LIN {X 0,Y 335.308,Z 623.747,A -85,B 0,C 180,E1 -19732.854,E2 -19732.854} C_VEL
LIN {X 0,Y 329.002,Z 618.791,A -85,B 0,C 180,E1 -19734.521,E2 -19734.521} C_VEL
LIN {X 0,Y 320.046,Z 611.53,A -85,B 0,C 180,E1 -19736.705,E2 -19736.705} C_VEL
LIN {X 0,Y 311.713,Z 604.517,A -85,B 0,C 180,E1 -19738.536,E2 -19738.536} C_VEL
LIN {X 0,Y 303.671,Z 597.573,A -85,B 0,C 180,E1 -19740.106,E2 -19740.106} C_VEL
LIN {X 0,Y 294.083,Z 589.042,A -85,B 0,C 180,E1 -19741.756,E2 -19741.756} C_VEL
LIN {X 0,Y 277.911,Z 573.415,A -85,B 0,C 180,E1 -19744.368,E2 -19744.368} C_VEL
LIN {X 0,Y 267.025,Z 560.92,A -85,B 0,C 180,E1 -19746.403,E2 -19746.403} C_VEL
LIN {X 0,Y 258.838,Z 549.026,A -85,B 0,C 180,E1 -19748.172,E2 -19748.172} C_VEL
LIN {X 0,Y 247.972,Z 530.618,A -85,B 0,C 180,E1 -19750.877,E2 -19750.877} C_VEL
LIN {X 0,Y 240.07,Z 518.715,A -85,B 0,C 180,E1 -19753.019,E2 -19753.019} C_VEL
LIN {X 0,Y 237.499,Z 514.891,A -85,B 0,C 180,E1 -19753.761,E2 -19753.761} C_VEL
LIN {X 0,Y 235.646,Z 512.583,A -85,B 0,C 180,E1 -19754.294,E2 -19754.294} C_VEL
LIN {X 0,Y 235.056,Z 510.889,A -85,B 0,C 180,E1 -19754.626,E2 -19754.626} C_VEL
LIN {X 0,Y 234.948,Z 510.343,A -85,B 0,C 180,E1 -19755.075,E2 -19755.075} C_VEL
LIN {X 0,Y 234.945,Z 510.328,A -85,B 0,C 180,E1 -19758.847,E2 -19758.847} C_VEL
LIN {X 0,Y 234.94,Z 510.326,A -85,B 0,C 180,E1 -19763.254,E2 -19763.254} C_VEL
LIN {X 0,Y 234.955,Z 510.335,A -85,B 0,C 180,E1 -19767.425,E2 -19767.425} C_VEL
LIN {X 0,Y 234.947,Z 510.334,A -85,B 0,C 180,E1 -19771.406,E2 -19771.406} C_VEL
LIN {X 0,Y 234.981,Z 510.31,A -85,B 0,C 180,E1 -19775.247,E2 -19775.247} C_VEL
LIN {X 0,Y 235.006,Z 510.337,A -85,B 0,C 180,E1 -19778.97,E2 -19778.97} C_VEL
LIN {X 0,Y 235.09,Z 510.293,A -85,B 0,C 180,E1 -19783.061,E2 -19783.061} C_VEL
LIN {X 0,Y 235.108,Z 510.307,A -85,B 0,C 180,E1 -19787.923,E2 -19787.923} C_VEL
LIN {X 0,Y 235.326,Z 510.265,A -85,B 0,C 180,E1 -19791.413,E2 -19791.413} C_VEL
LIN {X 0,Y 235.369,Z 510.285,A -85,B 0,C 180,E1 -19793.141,E2 -19793.141} C_VEL
LIN {X 0,Y 235.59,Z 510.222,A -85,B 0,C 180,E1 -19798.291,E2 -19798.291} C_VEL
LIN {X 0,Y 235.591,Z 510.26,A -85,B 0,C 180,E1 -19801.71,E2 -19801.71} C_VEL
LIN {X 0,Y 235.398,Z 510.252,A -85,B 0,C 180,E1 -19806.86,E2 -19806.86} C_VEL
LIN {X 0,Y 235.234,Z 510.306,A -85,B 0,C 180,E1 -19810.327,E2 -19810.327} C_VEL
LIN {X 0,Y 235.108,Z 510.306,A -85,B 0,C 180,E1 -19815.608,E2 -19815.608} C_VEL
LIN {X 0,Y 235.003,Z 510.313,A -85,B 0,C 180,E1 -19819.207,E2 -19819.207} C_VEL
LIN {X 0,Y 234.949,Z 510.333,A -85,B 0,C 180,E1 -19822.885,E2 -19822.885} C_VEL
LIN {X 0,Y 234.964,Z 510.315,A -85,B 0,C 180,E1 -19826.659,E2 -19826.659} C_VEL
LIN {X 0,Y 234.92,Z 510.347,A -85,B 0,C 180,E1 -19830.57,E2 -19830.57} C_VEL
LIN {X 0,Y 234.959,Z 510.33,A -85,B 0,C 180,E1 -19834.634,E2 -19834.634} C_VEL
LIN {X 0,Y 234.966,Z 510.331,A -85,B 0,C 180,E1 -19838.953,E2 -19838.953} C_VEL
LIN {X 0,Y 234.951,Z 510.537,A -85,B 0,C 180,E1 -19842.193,E2 -19842.193} C_VEL
LIN {X 0,Y 236.478,Z 516.25,A -85,B 0,C 180,E1 -19845.577,E2 -19845.577} C_VEL
LIN {X 0,Y 238.772,Z 520.508,A -85,B 0,C 180,E1 -19846.368,E2 -19846.368} C_VEL
LIN {X 0,Y 243.465,Z 528.613,A -85,B 0,C 180,E1 -19847.722,E2 -19847.722} C_VEL
LIN {X 0,Y 249.61,Z 540.017,A -85,B 0,C 180,E1 -19849.406,E2 -19849.406} C_VEL
LIN {X 0,Y 256.246,Z 553.836,A -85,B 0,C 180,E1 -19851.145,E2 -19851.145} C_VEL
LIN {X 0,Y 261.647,Z 566.971,A -85,B 0,C 180,E1 -19852.53,E2 -19852.53} C_VEL
LIN {X 0,Y 262.847,Z 573.625,A -85,B 0,C 180,E1 -19852.952,E2 -19852.952} C_VEL
LIN {X 0,Y 262.9,Z 576.826,A -85,B 0,C 180,E1 -19853.067,E2 -19853.067} C_VEL
LIN {X 0,Y 261.778,Z 581.327,A -85,B 0,C 180,E1 -19853.035,E2 -19853.035} C_VEL
LIN {X 0,Y 258.338,Z 590.232,A -85,B 0,C 180,E1 -19852.767,E2 -19852.767} C_VEL
LIN {X 0,Y 257.612,Z 594.257,A -85,B 0,C 180,E1 -19852.783,E2 -19852.783} C_VEL
LIN {X 0,Y 254.782,Z 653.012,A -85,B 0,C 180,E1 -19854.378,E2 -19854.378} C_VEL
LIN {X 0,Y 253.718,Z 664.354,A -85,B 0,C 180,E1 -19854.856,E2 -19854.856} C_VEL
LIN {X 0,Y 252.166,Z 675.789,A -85,B 0,C 180,E1 -19855.521,E2 -19855.521} C_VEL
LIN {X 0,Y 250.179,Z 687.439,A -85,B 0,C 180,E1 -19856.424,E2 -19856.424} C_VEL
LIN {X 0,Y 247.382,Z 701.15,A -85,B 0,C 180,E1 -19857.814,E2 -19857.814} C_VEL
LIN {X 0,Y 244.332,Z 713.482,A -85,B 0,C 180,E1 -19859.472,E2 -19859.472} C_VEL
LIN {X 0,Y 241.782,Z 723.247,A -85,B 0,C 180,E1 -19861.103,E2 -19861.103} C_VEL
LIN {X 0,Y 239.044,Z 732.264,A -85,B 0,C 180,E1 -19862.89,E2 -19862.89} C_VEL
LIN {X 0,Y 236.794,Z 739.236,A -85,B 0,C 180,E1 -19864.51,E2 -19864.51} C_VEL
LIN {X 0,Y 234.414,Z 746.76,A -85,B 0,C 180,E1 -19866.594,E2 -19866.594} C_VEL
LIN {X 0,Y 232.273,Z 753.234,A -85,B 0,C 180,E1 -19868.71,E2 -19868.71} C_VEL
LIN {X 0,Y 230.021,Z 760.213,A -85,B 0,C 180,E1 -19871.499,E2 -19871.499} C_VEL
LIN {X 0,Y 228.524,Z 765.213,A -85,B 0,C 180,E1 -19873.932,E2 -19873.932} C_VEL
LIN {X 0,Y 227.23,Z 769.661,A -85,B 0,C 180,E1 -19876.587,E2 -19876.587} C_VEL
LIN {X 0,Y 226.362,Z 773.212,A -85,B 0,C 180,E1 -19879.264,E2 -19879.264} C_VEL
LIN {X 0,Y 225.99,Z 775.156,A -85,B 0,C 180,E1 -19881.055,E2 -19881.055} C_VEL
LIN {X 0,Y 225.644,Z 777.85,A -85,B 0,C 180,E1 -19884.639,E2 -19884.639} C_VEL
LIN {X 0,Y 225.64,Z 779.149,A -85,B 0,C 180,E1 -19888.215,E2 -19888.215} C_VEL
LIN {X 0,Y 225.716,Z 779.404,A -85,B 0,C 180,E1 -19890,E2 -19890} C_VEL
LIN {X 0,Y 225.584,Z 778.671,A -85,B 0,C 180,E1 -19893.572,E2 -19893.572} C_VEL
LIN {X 0,Y 225.644,Z 777.85,A -85,B 0,C 180,E1 -19895.361,E2 -19895.361} C_VEL
LIN {X 0,Y 225.99,Z 775.156,A -85,B 0,C 180,E1 -19898.945,E2 -19898.945} C_VEL
LIN {X 0,Y 226.591,Z 772.193,A -85,B 0,C 180,E1 -19901.631,E2 -19901.631} C_VEL
LIN {X 0,Y 227.632,Z 768.363,A -85,B 0,C 180,E1 -19904.299,E2 -19904.299} C_VEL
LIN {X 0,Y 229.041,Z 763.597,A -85,B 0,C 180,E1 -19906.948,E2 -19906.948} C_VEL
LIN {X 0,Y 231.158,Z 756.648,A -85,B 0,C 180,E1 -19910.001,E2 -19910.001} C_VEL
LIN {X 0,Y 233.077,Z 750.772,A -85,B 0,C 180,E1 -19912.142,E2 -19912.142} C_VEL
LIN {X 0,Y 235.796,Z 742.36,A -85,B 0,C 180,E1 -19914.662,E2 -19914.662} C_VEL
LIN {X 0,Y 237.911,Z 735.901,A -85,B 0,C 180,E1 -19916.302,E2 -19916.302} C_VEL
LIN {X 0,Y 240.892,Z 726.426,A -85,B 0,C 180,E1 -19918.3,E2 -19918.3} C_VEL
LIN {X 0,Y 243.327,Z 717.587,A -85,B 0,C 180,E1 -19919.875,E2 -19919.875} C_VEL
LIN {X 0,Y 245.614,Z 708.498,A -85,B 0,C 180,E1 -19921.239,E2 -19921.239} C_VEL
LIN {X 0,Y 248.097,Z 697.694,A -85,B 0,C 180,E1 -19922.562,E2 -19922.562} C_VEL
LIN {X 0,Y 250.187,Z 687.44,A -85,B 0,C 180,E1 -19923.575,E2 -19923.575} C_VEL
LIN {X 0,Y 251.97,Z 677.149,A -85,B 0,C 180,E1 -19924.389,E2 -19924.389} C_VEL
LIN {X 0,Y 253.609,Z 665.266,A -85,B 0,C 180,E1 -19925.1,E2 -19925.1} C_VEL
LIN {X 0,Y 254.706,Z 653.918,A -85,B 0,C 180,E1 -19925.59,E2 -19925.59} C_VEL
LIN {X 0,Y 256.027,Z 629.639,A -85,B 0,C 180,E1 -19926.273,E2 -19926.273} C_VEL
LIN {X 0,Y 258.131,Z 580.661,A -85,B 0,C 180,E1 -19927.595,E2 -19927.595} C_VEL
LIN {X 0,Y 256.026,Z 569.105,A -85,B 0,C 180,E1 -19928.359,E2 -19928.359} C_VEL
LIN {X 0,Y 249.816,Z 554.326,A -85,B 0,C 180,E1 -19930.027,E2 -19930.027} C_VEL
LIN {X 0,Y 243.956,Z 542.258,A -85,B 0,C 180,E1 -19931.647,E2 -19931.647} C_VEL
LIN {X 0,Y 237.336,Z 529.983,A -85,B 0,C 180,E1 -19933.573,E2 -19933.573} C_VEL
LIN {X 0,Y 231.653,Z 520.434,A -85,B 0,C 180,E1 -19935.326,E2 -19935.326} C_VEL
LIN {X 0,Y 229.167,Z 516.078,A -85,B 0,C 180,E1 -19936.215,E2 -19936.215} C_VEL
LIN {X 0,Y 228.519,Z 513.68,A -85,B 0,C 180,E1 -19937.569,E2 -19937.569} C_VEL
LIN {X 0,Y 227.869,Z 511.239,A -85,B 0,C 180,E1 -19939.359,E2 -19939.359} C_VEL
LIN {X 0,Y 227.9,Z 511.223,A -85,B 0,C 180,E1 -19944.131,E2 -19944.131} C_VEL
LIN {X 0,Y 227.867,Z 511.211,A -85,B 0,C 180,E1 -19948.376,E2 -19948.376} C_VEL
LIN {X 0,Y 227.875,Z 511.196,A -85,B 0,C 180,E1 -19952.443,E2 -19952.443} C_VEL
LIN {X 0,Y 227.903,Z 511.221,A -85,B 0,C 180,E1 -19956.365,E2 -19956.365} C_VEL
LIN {X 0,Y 227.933,Z 511.187,A -85,B 0,C 180,E1 -19960.173,E2 -19960.173} C_VEL
LIN {X 0,Y 228.053,Z 511.194,A -85,B 0,C 180,E1 -19963.897,E2 -19963.897} C_VEL
LIN {X 0,Y 228.069,Z 511.167,A -85,B 0,C 180,E1 -19967.542,E2 -19967.542} C_VEL
LIN {X 0,Y 228.301,Z 511.167,A -85,B 0,C 180,E1 -19971.145,E2 -19971.145} C_VEL
LIN {X 0,Y 228.349,Z 511.132,A -85,B 0,C 180,E1 -19972.928,E2 -19972.928} C_VEL
LIN {X 0,Y 228.549,Z 511.138,A -85,B 0,C 180,E1 -19978.237,E2 -19978.237} C_VEL
LIN {X 0,Y 228.549,Z 511.098,A -85,B 0,C 180,E1 -19981.761,E2 -19981.761} C_VEL
LIN {X 0,Y 228.318,Z 511.16,A -85,B 0,C 180,E1 -19987.072,E2 -19987.072} C_VEL
LIN {X 0,Y 228.14,Z 511.155,A -85,B 0,C 180,E1 -19990.651,E2 -19990.651} C_VEL
LIN {X 0,Y 228.054,Z 511.201,A -85,B 0,C 180,E1 -19994.272,E2 -19994.272} C_VEL
LIN {X 0,Y 227.997,Z 511.176,A -85,B 0,C 180,E1 -19997.953,E2 -19997.953} C_VEL
LIN {X 0,Y 227.924,Z 511.204,A -85,B 0,C 180,E1 -20002.328,E2 -20002.328} C_VEL
LIN {X 0,Y 227.938,Z 511.208,A -85,B 0,C 180,E1 -20006.603,E2 -20006.603} C_VEL
LIN {X 0,Y 227.903,Z 511.194,A -85,B 0,C 180,E1 -20010.296,E2 -20010.296} C_VEL
LIN {X 0,Y 227.885,Z 511.223,A -85,B 0,C 180,E1 -20013.718,E2 -20013.718} C_VEL
LIN {X 0,Y 227.866,Z 511.223,A -85,B 0,C 180,E1 -20018.085,E2 -20018.085} C_VEL
LIN {X 0,Y 227.917,Z 511.218,A -85,B 0,C 180,E1 -20022.716,E2 -20022.716} C_VEL
LIN {X 0,Y 227.997,Z 511.569,A -85,B 0,C 180,E1 -20023.529,E2 -20023.529} C_VEL
LIN {X 0,Y 228.338,Z 512.86,A -85,B 0,C 180,E1 -20023.875,E2 -20023.875} C_VEL
LIN {X 0,Y 229.961,Z 515.367,A -85,B 0,C 180,E1 -20024.42,E2 -20024.42} C_VEL
LIN {X 0,Y 231.11,Z 516.52,A -85,B 0,C 180,E1 -20024.762,E2 -20024.762} C_VEL
LIN {X 0,Y 233.438,Z 520.082,A -85,B 0,C 180,E1 -20025.49,E2 -20025.49} C_VEL
LIN {X 0,Y 234.978,Z 522.293,A -85,B 0,C 180,E1 -20025.953,E2 -20025.953} C_VEL
LIN {X 0,Y 242.324,Z 533.357,A -85,B 0,C 180,E1 -20028.056,E2 -20028.056} C_VEL
LIN {X 0,Y 249.51,Z 545.346,A -85,B 0,C 180,E1 -20029.976,E2 -20029.976} C_VEL
LIN {X 0,Y 257.704,Z 559.01,A -85,B 0,C 180,E1 -20031.976,E2 -20031.976} C_VEL
LIN {X 0,Y 265.093,Z 568.867,A -85,B 0,C 180,E1 -20033.55,E2 -20033.55} C_VEL
LIN {X 0,Y 276.225,Z 581.407,A -85,B 0,C 180,E1 -20035.638,E2 -20035.638} C_VEL
LIN {X 0,Y 292.783,Z 596.955,A -85,B 0,C 180,E1 -20038.308,E2 -20038.308} C_VEL
LIN {X 0,Y 301.941,Z 604.909,A -85,B 0,C 180,E1 -20039.85,E2 -20039.85} C_VEL
LIN {X 0,Y 310.516,Z 612.189,A -85,B 0,C 180,E1 -20041.501,E2 -20041.501} C_VEL
LIN {X 0,Y 316.877,Z 617.435,A -85,B 0,C 180,E1 -20042.863,E2 -20042.863} C_VEL
LIN {X 0,Y 323.574,Z 622.734,A -85,B 0,C 180,E1 -20044.418,E2 -20044.418} C_VEL
LIN {X 0,Y 330.754,Z 628.529,A -85,B 0,C 180,E1 -20046.227,E2 -20046.227} C_VEL
LIN {X 0,Y 337.303,Z 633.472,A -85,B 0,C 180,E1 -20048.004,E2 -20048.004} C_VEL
LIN {X 0,Y 343.839,Z 638.407,A -85,B 0,C 180,E1 -20049.934,E2 -20049.934} C_VEL
LIN {X 0,Y 348.926,Z 641.956,A -85,B 0,C 180,E1 -20051.568,E2 -20051.568} C_VEL
LIN {X 0,Y 354.152,Z 646.014,A -85,B 0,C 180,E1 -20053.441,E2 -20053.441} C_VEL
LIN {X 0,Y 359.047,Z 649.045,A -85,B 0,C 180,E1 -20055.375,E2 -20055.375} C_VEL
LIN {X 0,Y 362.134,Z 650.902,A -85,B 0,C 180,E1 -20056.733,E2 -20056.733} C_VEL
LIN {X 0,Y 366.126,Z 654.139,A -85,B 0,C 180,E1 -20058.788,E2 -20058.788} C_VEL
LIN {X 0,Y 369.549,Z 656.326,A -85,B 0,C 180,E1 -20060.87,E2 -20060.87} C_VEL
LIN {X 0,Y 372.303,Z 657.773,A -85,B 0,C 180,E1 -20062.957,E2 -20062.957} C_VEL
LIN {X 0,Y 374.072,Z 658.637,A -85,B 0,C 180,E1 -20064.711,E2 -20064.711} C_VEL
LIN {X 0,Y 375.556,Z 659.129,A -85,B 0,C 180,E1 -20066.782,E2 -20066.782} C_VEL
LIN {X 0,Y 376.32,Z 659.56,A -85,B 0,C 180,E1 -20068.93,E2 -20068.93} C_VEL
LIN {X 0,Y 376.437,Z 659.445,A -85,B 0,C 180,E1 -20070,E2 -20070} C_VEL
LIN {X 0,Y 376.32,Z 659.564,A -85,B 0,C 180,E1 -20071.07,E2 -20071.07} C_VEL
LIN {X 0,Y 375.557,Z 659.127,A -85,B 0,C 180,E1 -20073.218,E2 -20073.218} C_VEL
LIN {X 0,Y 373.986,Z 658.612,A -85,B 0,C 180,E1 -20075.391,E2 -20075.391} C_VEL
LIN {X 0,Y 371.622,Z 657.459,A -85,B 0,C 180,E1 -20077.607,E2 -20077.607} C_VEL
LIN {X 0,Y 368.673,Z 655.793,A -85,B 0,C 180,E1 -20079.698,E2 -20079.698} C_VEL
LIN {X 0,Y 365.249,Z 653.465,A -85,B 0,C 180,E1 -20081.687,E2 -20081.687} C_VEL
LIN {X 0,Y 360.689,Z 649.881,A -85,B 0,C 180,E1 -20083.935,E2 -20083.935} C_VEL
LIN {X 0,Y 355.593,Z 646.933,A -85,B 0,C 180,E1 -20086.016,E2 -20086.016} C_VEL
LIN {X 0,Y 350.274,Z 643.071,A -85,B 0,C 180,E1 -20087.961,E2 -20087.961} C_VEL
LIN {X 0,Y 345.702,Z 639.604,A -85,B 0,C 180,E1 -20089.488,E2 -20089.488} C_VEL
LIN {X 0,Y 339.686,Z 635.398,A -85,B 0,C 180,E1 -20091.306,E2 -20091.306} C_VEL
LIN {X 0,Y 333.275,Z 630.389,A -85,B 0,C 180,E1 -20093.108,E2 -20093.108} C_VEL
LIN {X 0,Y 326.315,Z 624.983,A -85,B 0,C 180,E1 -20094.906,E2 -20094.906} C_VEL
LIN {X 0,Y 317.944,Z 618.316,A -85,B 0,C 180,E1 -20096.898,E2 -20096.898} C_VEL
LIN {X 0,Y 310.858,Z 612.45,A -85,B 0,C 180,E1 -20098.432,E2 -20098.432} C_VEL
LIN {X 0,Y 302.511,Z 605.374,A -85,B 0,C 180,E1 -20100.049,E2 -20100.049} C_VEL
LIN {X 0,Y 293.877,Z 597.842,A -85,B 0,C 180,E1 -20101.524,E2 -20101.524} C_VEL
LIN {X 0,Y 281.922,Z 587.013,A -85,B 0,C 180,E1 -20103.4,E2 -20103.4} C_VEL
LIN {X 0,Y 269.015,Z 573.605,A -85,B 0,C 180,E1 -20105.678,E2 -20105.678} C_VEL
LIN {X 0,Y 260.013,Z 562.278,A -85,B 0,C 180,E1 -20107.512,E2 -20107.512} C_VEL
LIN {X 0,Y 252.769,Z 551.145,A -85,B 0,C 180,E1 -20109.193,E2 -20109.193} C_VEL
LIN {X 0,Y 244.639,Z 537.086,A -85,B 0,C 180,E1 -20111.312,E2 -20111.312} C_VEL
LIN {X 0,Y 236.448,Z 524.329,A -85,B 0,C 180,E1 -20113.617,E2 -20113.617} C_VEL
LIN {X 0,Y 233.296,Z 519.919,A -85,B 0,C 180,E1 -20114.551,E2 -20114.551} C_VEL
LIN {X 0,Y 231.115,Z 516.466,A -85,B 0,C 180,E1 -20115.24,E2 -20115.24} C_VEL
LIN {X 0,Y 228.787,Z 513.771,A -85,B 0,C 180,E1 -20115.954,E2 -20115.954} C_VEL
LIN {X 0,Y 228.029,Z 511.698,A -85,B 0,C 180,E1 -20116.402,E2 -20116.402} C_VEL
LIN {X 0,Y 227.938,Z 511.24,A -85,B 0,C 180,E1 -20116.987,E2 -20116.987} C_VEL
LIN {X 0,Y 227.901,Z 511.211,A -85,B 0,C 180,E1 -20120.438,E2 -20120.438} C_VEL
LIN {X 0,Y 227.896,Z 511.201,A -85,B 0,C 180,E1 -20124.132,E2 -20124.132} C_VEL
LIN {X 0,Y 227.867,Z 511.204,A -85,B 0,C 180,E1 -20128.378,E2 -20128.378} C_VEL
LIN {X 0,Y 227.881,Z 511.226,A -85,B 0,C 180,E1 -20132.445,E2 -20132.445} C_VEL
LIN {X 0,Y 227.908,Z 511.191,A -85,B 0,C 180,E1 -20136.368,E2 -20136.368} C_VEL
LIN {X 0,Y 227.936,Z 511.207,A -85,B 0,C 180,E1 -20140.175,E2 -20140.175} C_VEL
LIN {X 0,Y 228.048,Z 511.175,A -85,B 0,C 180,E1 -20143.898,E2 -20143.898} C_VEL
LIN {X 0,Y 228.065,Z 511.189,A -85,B 0,C 180,E1 -20147.544,E2 -20147.544} C_VEL
LIN {X 0,Y 228.262,Z 511.141,A -85,B 0,C 180,E1 -20151.145,E2 -20151.145} C_VEL
LIN {X 0,Y 228.319,Z 511.16,A -85,B 0,C 180,E1 -20152.928,E2 -20152.928} C_VEL
LIN {X 0,Y 228.549,Z 511.098,A -85,B 0,C 180,E1 -20158.239,E2 -20158.239} C_VEL
LIN {X 0,Y 228.549,Z 511.138,A -85,B 0,C 180,E1 -20161.763,E2 -20161.763} C_VEL
LIN {X 0,Y 228.349,Z 511.132,A -85,B 0,C 180,E1 -20167.072,E2 -20167.072} C_VEL
LIN {X 0,Y 228.155,Z 511.184,A -85,B 0,C 180,E1 -20170.652,E2 -20170.652} C_VEL
LIN {X 0,Y 228.058,Z 511.167,A -85,B 0,C 180,E1 -20174.273,E2 -20174.273} C_VEL
LIN {X 0,Y 227.999,Z 511.204,A -85,B 0,C 180,E1 -20177.954,E2 -20177.954} C_VEL
LIN {X 0,Y 227.913,Z 511.199,A -85,B 0,C 180,E1 -20182.322,E2 -20182.322} C_VEL
LIN {X 0,Y 227.939,Z 511.189,A -85,B 0,C 180,E1 -20186.603,E2 -20186.603} C_VEL
LIN {X 0,Y 227.895,Z 511.224,A -85,B 0,C 180,E1 -20190.292,E2 -20190.292} C_VEL
LIN {X 0,Y 227.887,Z 511.201,A -85,B 0,C 180,E1 -20193.72,E2 -20193.72} C_VEL
LIN {X 0,Y 227.87,Z 511.21,A -85,B 0,C 180,E1 -20198.087,E2 -20198.087} C_VEL
LIN {X 0,Y 227.895,Z 511.419,A -85,B 0,C 180,E1 -20200.904,E2 -20200.904} C_VEL
LIN {X 0,Y 229.146,Z 515.969,A -85,B 0,C 180,E1 -20203.752,E2 -20203.752} C_VEL
LIN {X 0,Y 231.497,Z 520.231,A -85,B 0,C 180,E1 -20204.627,E2 -20204.627} C_VEL
LIN {X 0,Y 236.228,Z 528.091,A -85,B 0,C 180,E1 -20206.094,E2 -20206.094} C_VEL
LIN {X 0,Y 240.956,Z 536.487,A -85,B 0,C 180,E1 -20207.492,E2 -20207.492} C_VEL
LIN {X 0,Y 248.422,Z 551.234,A -85,B 0,C 180,E1 -20209.59,E2 -20209.59} C_VEL
LIN {X 0,Y 255.27,Z 567.143,A -85,B 0,C 180,E1 -20211.439,E2 -20211.439} C_VEL
LIN {X 0,Y 256.505,Z 571.097,A -85,B 0,C 180,E1 -20211.794,E2 -20211.794} C_VEL
LIN {X 0,Y 258.2,Z 581.48,A -85,B 0,C 180,E1 -20212.445,E2 -20212.445} C_VEL
LIN {X 0,Y 257.612,Z 594.257,A -85,B 0,C 180,E1 -20212.783,E2 -20212.783} C_VEL
LIN {X 0,Y 256.787,Z 600.112,A -85,B 0,C 180,E1 -20212.845,E2 -20212.845} C_VEL
LIN {X 0,Y 251.24,Z 619.14,A -85,B 0,C 180,E1 -20212.56,E2 -20212.56} C_VEL
LIN {X 0,Y 250.533,Z 624.985,A -85,B 0,C 180,E1 -20212.643,E2 -20212.643} C_VEL
LIN {X 0,Y 248.961,Z 653.984,A -85,B 0,C 180,E1 -20213.468,E2 -20213.468} C_VEL
LIN {X 0,Y 247.546,Z 667.804,A -85,B 0,C 180,E1 -20214.096,E2 -20214.096} C_VEL
LIN {X 0,Y 245.279,Z 681.875,A -85,B 0,C 180,E1 -20215.037,E2 -20215.037} C_VEL
LIN {X 0,Y 242.906,Z 693.989,A -85,B 0,C 180,E1 -20216.155,E2 -20216.155} C_VEL
LIN {X 0,Y 240.651,Z 703.907,A -85,B 0,C 180,E1 -20217.298,E2 -20217.298} C_VEL
LIN {X 0,Y 238.12,Z 713.631,A -85,B 0,C 180,E1 -20218.656,E2 -20218.656} C_VEL
LIN {X 0,Y 235.56,Z 723.048,A -85,B 0,C 180,E1 -20220.264,E2 -20220.264} C_VEL
LIN {X 0,Y 232.723,Z 732.066,A -85,B 0,C 180,E1 -20222.091,E2 -20222.091} C_VEL
LIN {X 0,Y 230.355,Z 739.036,A -85,B 0,C 180,E1 -20223.744,E2 -20223.744} C_VEL
LIN {X 0,Y 227.859,Z 746.56,A -85,B 0,C 180,E1 -20225.879,E2 -20225.879} C_VEL
LIN {X 0,Y 225.199,Z 754.172,A -85,B 0,C 180,E1 -20228.489,E2 -20228.489} C_VEL
LIN {X 0,Y 223.268,Z 759.765,A -85,B 0,C 180,E1 -20230.795,E2 -20230.795} C_VEL
LIN {X 0,Y 221.649,Z 765.013,A -85,B 0,C 180,E1 -20233.419,E2 -20233.419} C_VEL
LIN {X 0,Y 220.277,Z 769.462,A -85,B 0,C 180,E1 -20236.156,E2 -20236.156} C_VEL
LIN {X 0,Y 219.336,Z 773.012,A -85,B 0,C 180,E1 -20238.916,E2 -20238.916} C_VEL
LIN {X 0,Y 218.952,Z 774.957,A -85,B 0,C 180,E1 -20240.765,E2 -20240.765} C_VEL
LIN {X 0,Y 218.565,Z 777.652,A -85,B 0,C 180,E1 -20244.464,E2 -20244.464} C_VEL
LIN {X 0,Y 218.537,Z 778.951,A -85,B 0,C 180,E1 -20248.157,E2 -20248.157} C_VEL
LIN {X 0,Y 218.631,Z 779.206,A -85,B 0,C 180,E1 -20250,E2 -20250} C_VEL
LIN {X 0,Y 218.5,Z 778.473,A -85,B 0,C 180,E1 -20253.688,E2 -20253.688} C_VEL
LIN {X 0,Y 218.565,Z 777.652,A -85,B 0,C 180,E1 -20255.536,E2 -20255.536} C_VEL
LIN {X 0,Y 218.952,Z 774.957,A -85,B 0,C 180,E1 -20259.235,E2 -20259.235} C_VEL
LIN {X 0,Y 219.6,Z 771.994,A -85,B 0,C 180,E1 -20262.006,E2 -20262.006} C_VEL
LIN {X 0,Y 220.7,Z 768.163,A -85,B 0,C 180,E1 -20264.759,E2 -20264.759} C_VEL
LIN {X 0,Y 222.213,Z 763.397,A -85,B 0,C 180,E1 -20267.485,E2 -20267.485} C_VEL
LIN {X 0,Y 224.452,Z 756.448,A -85,B 0,C 180,E1 -20270.625,E2 -20270.625} C_VEL
LIN {X 0,Y 226.91,Z 749.235,A -85,B 0,C 180,E1 -20273.259,E2 -20273.259} C_VEL
LIN {X 0,Y 229.303,Z 742.16,A -85,B 0,C 180,E1 -20275.409,E2 -20275.409} C_VEL
LIN {X 0,Y 231.543,Z 735.702,A -85,B 0,C 180,E1 -20277.083,E2 -20277.083} C_VEL
LIN {X 0,Y 234.624,Z 726.227,A -85,B 0,C 180,E1 -20279.127,E2 -20279.127} C_VEL
LIN {X 0,Y 237.177,Z 717.257,A -85,B 0,C 180,E1 -20280.758,E2 -20280.758} C_VEL
LIN {X 0,Y 239.559,Z 708.299,A -85,B 0,C 180,E1 -20282.122,E2 -20282.122} C_VEL
LIN {X 0,Y 242.118,Z 697.495,A -85,B 0,C 180,E1 -20283.47,E2 -20283.47} C_VEL
LIN {X 0,Y 244.305,Z 687.242,A -85,B 0,C 180,E1 -20284.496,E2 -20284.496} C_VEL
LIN {X 0,Y 246.156,Z 676.952,A -85,B 0,C 180,E1 -20285.32,E2 -20285.32} C_VEL
LIN {X 0,Y 247.844,Z 665.068,A -85,B 0,C 180,E1 -20286.042,E2 -20286.042} C_VEL
LIN {X 0,Y 248.963,Z 653.931,A -85,B 0,C 180,E1 -20286.531,E2 -20286.531} C_VEL
LIN {X 0,Y 250.324,Z 629.85,A -85,B 0,C 180,E1 -20287.222,E2 -20287.222} C_VEL
LIN {X 0,Y 252.48,Z 581.797,A -85,B 0,C 180,E1 -20288.542,E2 -20288.542} C_VEL
LIN {X 0,Y 250.715,Z 571.982,A -85,B 0,C 180,E1 -20289.215,E2 -20289.215} C_VEL
LIN {X 0,Y 244.362,Z 556.878,A -85,B 0,C 180,E1 -20291.005,E2 -20291.005} C_VEL
LIN {X 0,Y 238.086,Z 543.913,A -85,B 0,C 180,E1 -20292.841,E2 -20292.841} C_VEL
LIN {X 0,Y 232.658,Z 533.911,A -85,B 0,C 180,E1 -20294.506,E2 -20294.506} C_VEL
LIN {X 0,Y 227.462,Z 525.127,A -85,B 0,C 180,E1 -20296.187,E2 -20296.187} C_VEL
LIN {X 0,Y 224.388,Z 520.144,A -85,B 0,C 180,E1 -20297.235,E2 -20297.235} C_VEL
LIN {X 0,Y 221.763,Z 515.684,A -85,B 0,C 180,E1 -20298.277,E2 -20298.277} C_VEL
LIN {X 0,Y 220.848,Z 512.158,A -85,B 0,C 180,E1 -20300.619,E2 -20300.619} C_VEL
LIN {X 0,Y 220.814,Z 512.095,A -85,B 0,C 180,E1 -20305.047,E2 -20305.047} C_VEL
LIN {X 0,Y 220.832,Z 512.101,A -85,B 0,C 180,E1 -20309.388,E2 -20309.388} C_VEL
LIN {X 0,Y 220.891,Z 512.067,A -85,B 0,C 180,E1 -20313.548,E2 -20313.548} C_VEL
LIN {X 0,Y 220.862,Z 512.078,A -85,B 0,C 180,E1 -20317.551,E2 -20317.551} C_VEL
LIN {X 0,Y 220.981,Z 512.083,A -85,B 0,C 180,E1 -20322.571,E2 -20322.571} C_VEL
LIN {X 0,Y 221.008,Z 512.043,A -85,B 0,C 180,E1 -20327.137,E2 -20327.137} C_VEL
LIN {X 0,Y 221.232,Z 512.051,A -85,B 0,C 180,E1 -20330.86,E2 -20330.86} C_VEL
LIN {X 0,Y 221.284,Z 512.014,A -85,B 0,C 180,E1 -20332.701,E2 -20332.701} C_VEL
LIN {X 0,Y 221.507,Z 512.015,A -85,B 0,C 180,E1 -20338.181,E2 -20338.181} C_VEL
LIN {X 0,Y 221.507,Z 511.974,A -85,B 0,C 180,E1 -20341.817,E2 -20341.817} C_VEL
LIN {X 0,Y 221.254,Z 512.037,A -85,B 0,C 180,E1 -20347.299,E2 -20347.299} C_VEL
LIN {X 0,Y 221.062,Z 512.038,A -85,B 0,C 180,E1 -20350.996,E2 -20350.996} C_VEL
LIN {X 0,Y 220.986,Z 512.075,A -85,B 0,C 180,E1 -20354.738,E2 -20354.738} C_VEL
LIN {X 0,Y 220.916,Z 512.061,A -85,B 0,C 180,E1 -20358.549,E2 -20358.549} C_VEL
LIN {X 0,Y 220.891,Z 512.073,A -85,B 0,C 180,E1 -20362.682,E2 -20362.682} C_VEL
LIN {X 0,Y 220.881,Z 512.094,A -85,B 0,C 180,E1 -20367.015,E2 -20367.015} C_VEL
LIN {X 0,Y 220.858,Z 512.072,A -85,B 0,C 180,E1 -20370.778,E2 -20370.778} C_VEL
LIN {X 0,Y 220.811,Z 512.087,A -85,B 0,C 180,E1 -20374.952,E2 -20374.952} C_VEL
LIN {X 0,Y 220.852,Z 512.089,A -85,B 0,C 180,E1 -20379.526,E2 -20379.526} C_VEL
LIN {X 0,Y 220.868,Z 512.335,A -85,B 0,C 180,E1 -20381.513,E2 -20381.513} C_VEL
LIN {X 0,Y 221.166,Z 513.443,A -85,B 0,C 180,E1 -20381.914,E2 -20381.914} C_VEL
LIN {X 0,Y 222.676,Z 516.001,A -85,B 0,C 180,E1 -20382.489,E2 -20382.489} C_VEL
LIN {X 0,Y 224.32,Z 517.645,A -85,B 0,C 180,E1 -20383.024,E2 -20383.024} C_VEL
LIN {X 0,Y 226.422,Z 520.935,A -85,B 0,C 180,E1 -20383.743,E2 -20383.743} C_VEL
LIN {X 0,Y 227.738,Z 522.621,A -85,B 0,C 180,E1 -20384.166,E2 -20384.166} C_VEL
LIN {X 0,Y 233.584,Z 531.193,A -85,B 0,C 180,E1 -20385.994,E2 -20385.994} C_VEL
LIN {X 0,Y 240.513,Z 542.081,A -85,B 0,C 180,E1 -20388.01,E2 -20388.01} C_VEL
LIN {X 0,Y 253.218,Z 563.727,A -85,B 0,C 180,E1 -20391.341,E2 -20391.341} C_VEL
LIN {X 0,Y 260.821,Z 573.983,A -85,B 0,C 180,E1 -20393.022,E2 -20393.022} C_VEL
LIN {X 0,Y 271.854,Z 586.561,A -85,B 0,C 180,E1 -20395.164,E2 -20395.164} C_VEL
LIN {X 0,Y 289.049,Z 602.771,A -85,B 0,C 180,E1 -20397.989,E2 -20397.989} C_VEL
LIN {X 0,Y 298.104,Z 610.541,A -85,B 0,C 180,E1 -20399.455,E2 -20399.455} C_VEL
LIN {X 0,Y 307.076,Z 617.983,A -85,B 0,C 180,E1 -20401.081,E2 -20401.081} C_VEL
LIN {X 0,Y 315.121,Z 624.561,A -85,B 0,C 180,E1 -20402.754,E2 -20402.754} C_VEL
LIN {X 0,Y 323.399,Z 631.047,A -85,B 0,C 180,E1 -20404.663,E2 -20404.663} C_VEL
LIN {X 0,Y 330.693,Z 636.677,A -85,B 0,C 180,E1 -20406.506,E2 -20406.506} C_VEL
LIN {X 0,Y 336.952,Z 641.459,A -85,B 0,C 180,E1 -20408.214,E2 -20408.214} C_VEL
LIN {X 0,Y 343.377,Z 646.009,A -85,B 0,C 180,E1 -20410.111,E2 -20410.111} C_VEL
LIN {X 0,Y 347.939,Z 649.276,A -85,B 0,C 180,E1 -20411.577,E2 -20411.577} C_VEL
LIN {X 0,Y 353.224,Z 653.209,A -85,B 0,C 180,E1 -20413.457,E2 -20413.457} C_VEL
LIN {X 0,Y 358.003,Z 656.101,A -85,B 0,C 180,E1 -20415.332,E2 -20415.332} C_VEL
LIN {X 0,Y 360.783,Z 657.77,A -85,B 0,C 180,E1 -20416.545,E2 -20416.545} C_VEL
LIN {X 0,Y 364.857,Z 661.023,A -85,B 0,C 180,E1 -20418.603,E2 -20418.603} C_VEL
LIN {X 0,Y 368.392,Z 663.262,A -85,B 0,C 180,E1 -20420.706,E2 -20420.706} C_VEL
LIN {X 0,Y 371.397,Z 664.821,A -85,B 0,C 180,E1 -20422.939,E2 -20422.939} C_VEL
LIN {X 0,Y 373.102,Z 665.649,A -85,B 0,C 180,E1 -20424.596,E2 -20424.596} C_VEL
LIN {X 0,Y 374.684,Z 666.176,A -85,B 0,C 180,E1 -20426.774,E2 -20426.774} C_VEL
LIN {X 0,Y 375.454,Z 666.604,A -85,B 0,C 180,E1 -20428.927,E2 -20428.927} C_VEL
LIN {X 0,Y 375.572,Z 666.489,A -85,B 0,C 180,E1 -20430,E2 -20430} C_VEL
LIN {X 0,Y 375.454,Z 666.61,A -85,B 0,C 180,E1 -20431.073,E2 -20431.073} C_VEL
LIN {X 0,Y 374.685,Z 666.173,A -85,B 0,C 180,E1 -20433.226,E2 -20433.226} C_VEL
LIN {X 0,Y 373.102,Z 665.655,A -85,B 0,C 180,E1 -20435.404,E2 -20435.404} C_VEL
LIN {X 0,Y 370.963,Z 664.676,A -85,B 0,C 180,E1 -20437.413,E2 -20437.413} C_VEL
LIN {X 0,Y 368.025,Z 663.006,A -85,B 0,C 180,E1 -20439.534,E2 -20439.534} C_VEL
LIN {X 0,Y 364.395,Z 660.675,A -85,B 0,C 180,E1 -20441.649,E2 -20441.649} C_VEL
LIN {X 0,Y 359.97,Z 657.106,A -85,B 0,C 180,E1 -20443.838,E2 -20443.838} C_VEL
LIN {X 0,Y 355.103,Z 654.406,A -85,B 0,C 180,E1 -20445.836,E2 -20445.836} C_VEL
LIN {X 0,Y 349.919,Z 650.815,A -85,B 0,C 180,E1 -20447.738,E2 -20447.738} C_VEL
LIN {X 0,Y 343.814,Z 646.237,A -85,B 0,C 180,E1 -20449.754,E2 -20449.754} C_VEL
LIN {X 0,Y 337.786,Z 642.087,A -85,B 0,C 180,E1 -20451.55,E2 -20451.55} C_VEL
LIN {X 0,Y 330.92,Z 636.809,A -85,B 0,C 180,E1 -20453.435,E2 -20453.435} C_VEL
LIN {X 0,Y 323.937,Z 631.473,A -85,B 0,C 180,E1 -20455.204,E2 -20455.204} C_VEL
LIN {X 0,Y 315.587,Z 624.943,A -85,B 0,C 180,E1 -20457.14,E2 -20457.14} C_VEL
LIN {X 0,Y 307.677,Z 618.488,A -85,B 0,C 180,E1 -20458.801,E2 -20458.801} C_VEL
LIN {X 0,Y 298.442,Z 610.833,A -85,B 0,C 180,E1 -20460.489,E2 -20460.489} C_VEL
LIN {X 0,Y 289.05,Z 602.766,A -85,B 0,C 180,E1 -20462.012,E2 -20462.012} C_VEL
LIN {X 0,Y 271.728,Z 586.427,A -85,B 0,C 180,E1 -20464.859,E2 -20464.859} C_VEL
LIN {X 0,Y 260.466,Z 573.566,A -85,B 0,C 180,E1 -20467.051,E2 -20467.051} C_VEL
LIN {X 0,Y 252.553,Z 562.75,A -85,B 0,C 180,E1 -20468.816,E2 -20468.816} C_VEL
LIN {X 0,Y 239.266,Z 540.014,A -85,B 0,C 180,E1 -20472.344,E2 -20472.344} C_VEL
LIN {X 0,Y 231.915,Z 528.709,A -85,B 0,C 180,E1 -20474.514,E2 -20474.514} C_VEL
LIN {X 0,Y 229.033,Z 524.59,A -85,B 0,C 180,E1 -20475.413,E2 -20475.413} C_VEL
LIN {X 0,Y 226.756,Z 521.28,A -85,B 0,C 180,E1 -20476.152,E2 -20476.152} C_VEL
LIN {X 0,Y 224.447,Z 517.959,A -85,B 0,C 180,E1 -20476.927,E2 -20476.927} C_VEL
LIN {X 0,Y 223.549,Z 516.816,A -85,B 0,C 180,E1 -20477.228,E2 -20477.228} C_VEL
LIN {X 0,Y 221.658,Z 514.585,A -85,B 0,C 180,E1 -20477.869,E2 -20477.869} C_VEL
LIN {X 0,Y 220.935,Z 512.607,A -85,B 0,C 180,E1 -20478.325,E2 -20478.325} C_VEL
LIN {X 0,Y 220.827,Z 512.101,A -85,B 0,C 180,E1 -20479.008,E2 -20479.008} C_VEL
LIN {X 0,Y 220.829,Z 512.087,A -85,B 0,C 180,E1 -20482.795,E2 -20482.795} C_VEL
LIN {X 0,Y 220.819,Z 512.097,A -85,B 0,C 180,E1 -20487.246,E2 -20487.246} C_VEL
LIN {X 0,Y 220.832,Z 512.091,A -85,B 0,C 180,E1 -20491.487,E2 -20491.487} C_VEL
LIN {X 0,Y 220.862,Z 512.066,A -85,B 0,C 180,E1 -20495.565,E2 -20495.565} C_VEL
LIN {X 0,Y 220.887,Z 512.094,A -85,B 0,C 180,E1 -20499.514,E2 -20499.514} C_VEL
LIN {X 0,Y 221.009,Z 512.047,A -85,B 0,C 180,E1 -20503.371,E2 -20503.371} C_VEL
LIN {X 0,Y 221.004,Z 512.075,A -85,B 0,C 180,E1 -20507.139,E2 -20507.139} C_VEL
LIN {X 0,Y 221.199,Z 512.018,A -85,B 0,C 180,E1 -20510.86,E2 -20510.86} C_VEL
LIN {X 0,Y 221.137,Z 512.059,A -85,B 0,C 180,E1 -20514.53,E2 -20514.53} C_VEL
LIN {X 0,Y 221.507,Z 511.974,A -85,B 0,C 180,E1 -20518.183,E2 -20518.183} C_VEL
LIN {X 0,Y 221.507,Z 512.015,A -85,B 0,C 180,E1 -20521.819,E2 -20521.819} C_VEL
LIN {X 0,Y 221.284,Z 512.014,A -85,B 0,C 180,E1 -20527.299,E2 -20527.299} C_VEL
LIN {X 0,Y 221.103,Z 512.055,A -85,B 0,C 180,E1 -20530.995,E2 -20530.995} C_VEL
LIN {X 0,Y 221.012,Z 512.077,A -85,B 0,C 180,E1 -20536.631,E2 -20536.631} C_VEL
LIN {X 0,Y 220.881,Z 512.062,A -85,B 0,C 180,E1 -20540.488,E2 -20540.488} C_VEL
LIN {X 0,Y 220.859,Z 512.097,A -85,B 0,C 180,E1 -20544.437,E2 -20544.437} C_VEL
LIN {X 0,Y 220.824,Z 512.081,A -85,B 0,C 180,E1 -20548.516,E2 -20548.516} C_VEL
LIN {X 0,Y 220.821,Z 512.079,A -85,B 0,C 180,E1 -20552.756,E2 -20552.756} C_VEL
LIN {X 0,Y 220.837,Z 512.087,A -85,B 0,C 180,E1 -20557.289,E2 -20557.289} C_VEL
LIN {X 0,Y 220.875,Z 512.289,A -85,B 0,C 180,E1 -20559.523,E2 -20559.523} C_VEL
LIN {X 0,Y 221.763,Z 515.683,A -85,B 0,C 180,E1 -20561.723,E2 -20561.723} C_VEL
LIN {X 0,Y 224.264,Z 519.977,A -85,B 0,C 180,E1 -20562.724,E2 -20562.724} C_VEL
LIN {X 0,Y 226.13,Z 523.02,A -85,B 0,C 180,E1 -20563.367,E2 -20563.367} C_VEL
LIN {X 0,Y 229.067,Z 527.8,A -85,B 0,C 180,E1 -20564.344,E2 -20564.344} C_VEL
LIN {X 0,Y 234.244,Z 536.668,A -85,B 0,C 180,E1 -20565.987,E2 -20565.987} C_VEL
LIN {X 0,Y 240.814,Z 549.32,A -85,B 0,C 180,E1 -20567.966,E2 -20567.966} C_VEL
LIN {X 0,Y 247.12,Z 563.175,A -85,B 0,C 180,E1 -20569.78,E2 -20569.78} C_VEL
LIN {X 0,Y 250.992,Z 572.956,A -85,B 0,C 180,E1 -20570.871,E2 -20570.871} C_VEL
LIN {X 0,Y 252.529,Z 582.474,A -85,B 0,C 180,E1 -20571.491,E2 -20571.491} C_VEL
LIN {X 0,Y 250.533,Z 624.985,A -85,B 0,C 180,E1 -20572.643,E2 -20572.643} C_VEL
LIN {X 0,Y 249.828,Z 630.831,A -85,B 0,C 180,E1 -20572.724,E2 -20572.724} C_VEL
LIN {X 0,Y 247.074,Z 640.34,A -85,B 0,C 180,E1 -20572.583,E2 -20572.583} C_VEL
LIN {X 0,Y 244.15,Z 649.834,A -85,B 0,C 180,E1 -20572.429,E2 -20572.429} C_VEL
LIN {X 0,Y 243.173,Z 655.664,A -85,B 0,C 180,E1 -20572.544,E2 -20572.544} C_VEL
LIN {X 0,Y 241.299,Z 671.316,A -85,B 0,C 180,E1 -20573.34,E2 -20573.34} C_VEL
LIN {X 0,Y 239.272,Z 682.749,A -85,B 0,C 180,E1 -20574.155,E2 -20574.155} C_VEL
LIN {X 0,Y 237.023,Z 693.791,A -85,B 0,C 180,E1 -20575.196,E2 -20575.196} C_VEL
LIN {X 0,Y 234.7,Z 703.709,A -85,B 0,C 180,E1 -20576.361,E2 -20576.361} C_VEL
LIN {X 0,Y 232.055,Z 713.432,A -85,B 0,C 180,E1 -20577.74,E2 -20577.74} C_VEL
LIN {X 0,Y 229.336,Z 722.865,A -85,B 0,C 180,E1 -20579.376,E2 -20579.376} C_VEL
LIN {X 0,Y 226.457,Z 731.867,A -85,B 0,C 180,E1 -20581.248,E2 -20581.248} C_VEL
LIN {X 0,Y 223.983,Z 738.837,A -85,B 0,C 180,E1 -20582.938,E2 -20582.938} C_VEL
LIN {X 0,Y 221.348,Z 746.361,A -85,B 0,C 180,E1 -20585.122,E2 -20585.122} C_VEL
LIN {X 0,Y 218.992,Z 752.834,A -85,B 0,C 180,E1 -20587.35,E2 -20587.35} C_VEL
LIN {X 0,Y 216.66,Z 759.305,A -85,B 0,C 180,E1 -20590.05,E2 -20590.05} C_VEL
LIN {X 0,Y 214.801,Z 764.814,A -85,B 0,C 180,E1 -20592.875,E2 -20592.875} C_VEL
LIN {X 0,Y 213.342,Z 769.262,A -85,B 0,C 180,E1 -20595.696,E2 -20595.696} C_VEL
LIN {X 0,Y 212.331,Z 772.813,A -85,B 0,C 180,E1 -20598.545,E2 -20598.545} C_VEL
LIN {X 0,Y 211.897,Z 774.758,A -85,B 0,C 180,E1 -20600.454,E2 -20600.454} C_VEL
LIN {X 0,Y 211.485,Z 777.454,A -85,B 0,C 180,E1 -20604.279,E2 -20604.279} C_VEL
LIN {X 0,Y 211.439,Z 778.753,A -85,B 0,C 180,E1 -20608.095,E2 -20608.095} C_VEL
LIN {X 0,Y 211.547,Z 779.009,A -85,B 0,C 180,E1 -20610,E2 -20610} C_VEL
LIN {X 0,Y 211.421,Z 778.091,A -85,B 0,C 180,E1 -20614.241,E2 -20614.241} C_VEL
LIN {X 0,Y 211.613,Z 776.217,A -85,B 0,C 180,E1 -20617.634,E2 -20617.634} C_VEL
LIN {X 0,Y 211.897,Z 774.758,A -85,B 0,C 180,E1 -20619.546,E2 -20619.546} C_VEL
LIN {X 0,Y 212.6,Z 771.794,A -85,B 0,C 180,E1 -20622.408,E2 -20622.408} C_VEL
LIN {X 0,Y 213.791,Z 767.964,A -85,B 0,C 180,E1 -20625.247,E2 -20625.247} C_VEL
LIN {X 0,Y 215.4,Z 763.198,A -85,B 0,C 180,E1 -20628.057,E2 -20628.057} C_VEL
LIN {X 0,Y 217.756,Z 756.248,A -85,B 0,C 180,E1 -20631.29,E2 -20631.29} C_VEL
LIN {X 0,Y 220.365,Z 749.036,A -85,B 0,C 180,E1 -20633.993,E2 -20633.993} C_VEL
LIN {X 0,Y 222.861,Z 741.96,A -85,B 0,C 180,E1 -20636.199,E2 -20636.199} C_VEL
LIN {X 0,Y 225.828,Z 733.685,A -85,B 0,C 180,E1 -20638.332,E2 -20638.332} C_VEL
LIN {X 0,Y 228.709,Z 724.968,A -85,B 0,C 180,E1 -20640.21,E2 -20640.21} C_VEL
LIN {X 0,Y 231.242,Z 716.535,A -85,B 0,C 180,E1 -20641.745,E2 -20641.745} C_VEL
LIN {X 0,Y 233.937,Z 706.637,A -85,B 0,C 180,E1 -20643.248,E2 -20643.248} C_VEL
LIN {X 0,Y 236.219,Z 697.297,A -85,B 0,C 180,E1 -20644.421,E2 -20644.421} C_VEL
LIN {X 0,Y 238.498,Z 687.044,A -85,B 0,C 180,E1 -20645.46,E2 -20645.46} C_VEL
LIN {X 0,Y 240.4,Z 676.754,A -85,B 0,C 180,E1 -20646.298,E2 -20646.298} C_VEL
LIN {X 0,Y 242.132,Z 664.87,A -85,B 0,C 180,E1 -20647.032,E2 -20647.032} C_VEL
LIN {X 0,Y 243.272,Z 653.949,A -85,B 0,C 180,E1 -20647.52,E2 -20647.52} C_VEL
LIN {X 0,Y 244.641,Z 631.434,A -85,B 0,C 180,E1 -20648.175,E2 -20648.175} C_VEL
LIN {X 0,Y 246.912,Z 583.102,A -85,B 0,C 180,E1 -20649.523,E2 -20649.523} C_VEL
LIN {X 0,Y 245.39,Z 574.729,A -85,B 0,C 180,E1 -20650.127,E2 -20650.127} C_VEL
LIN {X 0,Y 238.852,Z 559.033,A -85,B 0,C 180,E1 -20652.071,E2 -20652.071} C_VEL
LIN {X 0,Y 231.487,Z 544.069,A -85,B 0,C 180,E1 -20654.357,E2 -20654.357} C_VEL
LIN {X 0,Y 226.002,Z 534.294,A -85,B 0,C 180,E1 -20656.16,E2 -20656.16} C_VEL
LIN {X 0,Y 223.125,Z 529.49,A -85,B 0,C 180,E1 -20657.15,E2 -20657.15} C_VEL
LIN {X 0,Y 220.425,Z 525.021,A -85,B 0,C 180,E1 -20658.119,E2 -20658.119} C_VEL
LIN {X 0,Y 217.247,Z 520.048,A -85,B 0,C 180,E1 -20659.302,E2 -20659.302} C_VEL
LIN {X 0,Y 214.709,Z 515.979,A -85,B 0,C 180,E1 -20660.335,E2 -20660.335} C_VEL
LIN {X 0,Y 214.269,Z 514.753,A -85,B 0,C 180,E1 -20660.846,E2 -20660.846} C_VEL
LIN {X 0,Y 213.798,Z 513.008,A -85,B 0,C 180,E1 -20662.252,E2 -20662.252} C_VEL
LIN {X 0,Y 213.767,Z 512.961,A -85,B 0,C 180,E1 -20666.019,E2 -20666.019} C_VEL
LIN {X 0,Y 213.758,Z 512.976,A -85,B 0,C 180,E1 -20670.45,E2 -20670.45} C_VEL
LIN {X 0,Y 213.795,Z 512.963,A -85,B 0,C 180,E1 -20674.7,E2 -20674.7} C_VEL
LIN {X 0,Y 213.799,Z 512.944,A -85,B 0,C 180,E1 -20678.801,E2 -20678.801} C_VEL
LIN {X 0,Y 213.94,Z 512.961,A -85,B 0,C 180,E1 -20682.802,E2 -20682.802} C_VEL
LIN {X 0,Y 213.949,Z 512.92,A -85,B 0,C 180,E1 -20686.705,E2 -20686.705} C_VEL
LIN {X 0,Y 214.164,Z 512.933,A -85,B 0,C 180,E1 -20690.555,E2 -20690.555} C_VEL
LIN {X 0,Y 214.222,Z 512.896,A -85,B 0,C 180,E1 -20692.459,E2 -20692.459} C_VEL
LIN {X 0,Y 214.441,Z 512.896,A -85,B 0,C 180,E1 -20698.121,E2 -20698.121} C_VEL
LIN {X 0,Y 214.545,Z 512.858,A -85,B 0,C 180,E1 -20699.999,E2 -20699.999} C_VEL
LIN {X 0,Y 214.44,Z 512.854,A -85,B 0,C 180,E1 -20701.877,E2 -20701.877} C_VEL
LIN {X 0,Y 214.193,Z 512.91,A -85,B 0,C 180,E1 -20707.541,E2 -20707.541} C_VEL
LIN {X 0,Y 213.994,Z 512.922,A -85,B 0,C 180,E1 -20711.364,E2 -20711.364} C_VEL
LIN {X 0,Y 213.924,Z 512.945,A -85,B 0,C 180,E1 -20715.237,E2 -20715.237} C_VEL
LIN {X 0,Y 213.834,Z 512.95,A -85,B 0,C 180,E1 -20719.187,E2 -20719.187} C_VEL
LIN {X 0,Y 213.842,Z 512.945,A -85,B 0,C 180,E1 -20723.227,E2 -20723.227} C_VEL
LIN {X 0,Y 213.824,Z 512.976,A -85,B 0,C 180,E1 -20727.449,E2 -20727.449} C_VEL
LIN {X 0,Y 213.775,Z 512.959,A -85,B 0,C 180,E1 -20731.735,E2 -20731.735} C_VEL
LIN {X 0,Y 213.749,Z 512.962,A -85,B 0,C 180,E1 -20736.286,E2 -20736.286} C_VEL
LIN {X 0,Y 213.838,Z 513.225,A -85,B 0,C 180,E1 -20739.398,E2 -20739.398} C_VEL
LIN {X 0,Y 214.112,Z 514.307,A -85,B 0,C 180,E1 -20739.795,E2 -20739.795} C_VEL
LIN {X 0,Y 215.573,Z 516.845,A -85,B 0,C 180,E1 -20740.413,E2 -20740.413} C_VEL
LIN {X 0,Y 217.437,Z 518.659,A -85,B 0,C 180,E1 -20741.08,E2 -20741.08} C_VEL
LIN {X 0,Y 219.52,Z 521.878,A -85,B 0,C 180,E1 -20741.859,E2 -20741.859} C_VEL
LIN {X 0,Y 220.944,Z 523.601,A -85,B 0,C 180,E1 -20742.354,E2 -20742.354} C_VEL
LIN {X 0,Y 229.011,Z 535.21,A -85,B 0,C 180,E1 -20745.046,E2 -20745.046} C_VEL
LIN {X 0,Y 237.662,Z 549.172,A -85,B 0,C 180,E1 -20747.669,E2 -20747.669} C_VEL
LIN {X 0,Y 248.418,Z 567.931,A -85,B 0,C 180,E1 -20750.598,E2 -20750.598} C_VEL
LIN {X 0,Y 256.322,Z 578.843,A -85,B 0,C 180,E1 -20752.424,E2 -20752.424} C_VEL
LIN {X 0,Y 267.81,Z 592.011,A -85,B 0,C 180,E1 -20754.731,E2 -20754.731} C_VEL
LIN {X 0,Y 285.163,Z 608.497,A -85,B 0,C 180,E1 -20757.662,E2 -20757.662} C_VEL
LIN {X 0,Y 295.626,Z 617.303,A -85,B 0,C 180,E1 -20759.294,E2 -20759.294} C_VEL
LIN {X 0,Y 304.042,Z 624.229,A -85,B 0,C 180,E1 -20760.788,E2 -20760.788} C_VEL
LIN {X 0,Y 311.506,Z 630.126,A -85,B 0,C 180,E1 -20762.252,E2 -20762.252} C_VEL
LIN {X 0,Y 319.567,Z 636.299,A -85,B 0,C 180,E1 -20764.028,E2 -20764.028} C_VEL
LIN {X 0,Y 326.382,Z 641.684,A -85,B 0,C 180,E1 -20765.691,E2 -20765.691} C_VEL
LIN {X 0,Y 333.228,Z 646.767,A -85,B 0,C 180,E1 -20767.482,E2 -20767.482} C_VEL
LIN {X 0,Y 340.086,Z 651.778,A -85,B 0,C 180,E1 -20769.433,E2 -20769.433} C_VEL
LIN {X 0,Y 345.271,Z 655.312,A -85,B 0,C 180,E1 -20771.037,E2 -20771.037} C_VEL
LIN {X 0,Y 350.878,Z 659.514,A -85,B 0,C 180,E1 -20772.972,E2 -20772.972} C_VEL
LIN {X 0,Y 355.796,Z 662.545,A -85,B 0,C 180,E1 -20774.847,E2 -20774.847} C_VEL
LIN {X 0,Y 359.362,Z 664.598,A -85,B 0,C 180,E1 -20776.347,E2 -20776.347} C_VEL
LIN {X 0,Y 363.443,Z 667.852,A -85,B 0,C 180,E1 -20778.393,E2 -20778.393} C_VEL
LIN {X 0,Y 367.055,Z 670.156,A -85,B 0,C 180,E1 -20780.524,E2 -20780.524} C_VEL
LIN {X 0,Y 369.991,Z 671.686,A -85,B 0,C 180,E1 -20782.636,E2 -20782.636} C_VEL
LIN {X 0,Y 372.052,Z 672.67,A -85,B 0,C 180,E1 -20784.581,E2 -20784.581} C_VEL
LIN {X 0,Y 373.66,Z 673.175,A -85,B 0,C 180,E1 -20786.765,E2 -20786.765} C_VEL
LIN {X 0,Y 374.41,Z 673.626,A -85,B 0,C 180,E1 -20788.924,E2 -20788.924} C_VEL
LIN {X 0,Y 374.531,Z 673.513,A -85,B 0,C 180,E1 -20790,E2 -20790} C_VEL
LIN {X 0,Y 374.406,Z 673.631,A -85,B 0,C 180,E1 -20791.076,E2 -20791.076} C_VEL
LIN {X 0,Y 373.651,Z 673.175,A -85,B 0,C 180,E1 -20793.235,E2 -20793.235} C_VEL
LIN {X 0,Y 372.062,Z 672.666,A -85,B 0,C 180,E1 -20795.419,E2 -20795.419} C_VEL
LIN {X 0,Y 369.633,Z 671.543,A -85,B 0,C 180,E1 -20797.648,E2 -20797.648} C_VEL
LIN {X 0,Y 366.67,Z 669.864,A -85,B 0,C 180,E1 -20799.752,E2 -20799.752} C_VEL
LIN {X 0,Y 362.947,Z 667.486,A -85,B 0,C 180,E1 -20801.874,E2 -20801.874} C_VEL
LIN {X 0,Y 358.568,Z 663.965,A -85,B 0,C 180,E1 -20804.019,E2 -20804.019} C_VEL
LIN {X 0,Y 353.189,Z 660.991,A -85,B 0,C 180,E1 -20806.175,E2 -20806.175} C_VEL
LIN {X 0,Y 347.646,Z 657.163,A -85,B 0,C 180,E1 -20808.17,E2 -20808.17} C_VEL
LIN {X 0,Y 342.003,Z 652.959,A -85,B 0,C 180,E1 -20809.999,E2 -20809.999} C_VEL
LIN {X 0,Y 335.857,Z 648.777,A -85,B 0,C 180,E1 -20811.788,E2 -20811.788} C_VEL
LIN {X 0,Y 328.476,Z 643.22,A -85,B 0,C 180,E1 -20813.777,E2 -20813.777} C_VEL
LIN {X 0,Y 321.179,Z 637.652,A -85,B 0,C 180,E1 -20815.585,E2 -20815.585} C_VEL
LIN {X 0,Y 312.539,Z 630.973,A -85,B 0,C 180,E1 -20817.538,E2 -20817.538} C_VEL
LIN {X 0,Y 304.81,Z 624.831,A -85,B 0,C 180,E1 -20819.069,E2 -20819.069} C_VEL
LIN {X 0,Y 297.576,Z 618.843,A -85,B 0,C 180,E1 -20820.372,E2 -20820.372} C_VEL
LIN {X 0,Y 289.446,Z 612.165,A -85,B 0,C 180,E1 -20821.686,E2 -20821.686} C_VEL
LIN {X 0,Y 274.611,Z 598.774,A -85,B 0,C 180,E1 -20824.054,E2 -20824.054} C_VEL
LIN {X 0,Y 263.61,Z 587.387,A -85,B 0,C 180,E1 -20826.075,E2 -20826.075} C_VEL
LIN {X 0,Y 253.587,Z 575.39,A -85,B 0,C 180,E1 -20828.178,E2 -20828.178} C_VEL
LIN {X 0,Y 245.678,Z 563.462,A -85,B 0,C 180,E1 -20830.1,E2 -20830.1} C_VEL
LIN {X 0,Y 235.207,Z 545.039,A -85,B 0,C 180,E1 -20833.051,E2 -20833.051} C_VEL
LIN {X 0,Y 226.366,Z 531.238,A -85,B 0,C 180,E1 -20835.808,E2 -20835.808} C_VEL
LIN {X 0,Y 220.701,Z 523.151,A -85,B 0,C 180,E1 -20837.737,E2 -20837.737} C_VEL
LIN {X 0,Y 217.85,Z 519.515,A -85,B 0,C 180,E1 -20838.753,E2 -20838.753} C_VEL
LIN {X 0,Y 217.116,Z 518.125,A -85,B 0,C 180,E1 -20839.045,E2 -20839.045} C_VEL
LIN {X 0,Y 214.981,Z 516.08,A -85,B 0,C 180,E1 -20839.814,E2 -20839.814} C_VEL
LIN {X 0,Y 213.94,Z 513.595,A -85,B 0,C 180,E1 -20840.396,E2 -20840.396} C_VEL
LIN {X 0,Y 213.794,Z 512.997,A -85,B 0,C 180,E1 -20841.048,E2 -20841.048} C_VEL
LIN {X 0,Y 213.765,Z 512.976,A -85,B 0,C 180,E1 -20846.021,E2 -20846.021} C_VEL
LIN {X 0,Y 213.776,Z 512.957,A -85,B 0,C 180,E1 -20850.454,E2 -20850.454} C_VEL
LIN {X 0,Y 213.796,Z 512.95,A -85,B 0,C 180,E1 -20854.702,E2 -20854.702} C_VEL
LIN {X 0,Y 213.808,Z 512.977,A -85,B 0,C 180,E1 -20858.804,E2 -20858.804} C_VEL
LIN {X 0,Y 213.938,Z 512.924,A -85,B 0,C 180,E1 -20862.804,E2 -20862.804} C_VEL
LIN {X 0,Y 213.945,Z 512.959,A -85,B 0,C 180,E1 -20866.707,E2 -20866.707} C_VEL
LIN {X 0,Y 214.137,Z 512.896,A -85,B 0,C 180,E1 -20870.556,E2 -20870.556} C_VEL
LIN {X 0,Y 214.097,Z 512.937,A -85,B 0,C 180,E1 -20874.349,E2 -20874.349} C_VEL
LIN {X 0,Y 214.441,Z 512.854,A -85,B 0,C 180,E1 -20878.123,E2 -20878.123} C_VEL
LIN {X 0,Y 214.545,Z 512.858,A -85,B 0,C 180,E1 -20880.001,E2 -20880.001} C_VEL
LIN {X 0,Y 214.441,Z 512.896,A -85,B 0,C 180,E1 -20881.879,E2 -20881.879} C_VEL
LIN {X 0,Y 214.222,Z 512.896,A -85,B 0,C 180,E1 -20887.541,E2 -20887.541} C_VEL
LIN {X 0,Y 214.019,Z 512.929,A -85,B 0,C 180,E1 -20891.364,E2 -20891.364} C_VEL
LIN {X 0,Y 213.927,Z 512.935,A -85,B 0,C 180,E1 -20895.238,E2 -20895.238} C_VEL
LIN {X 0,Y 213.832,Z 512.948,A -85,B 0,C 180,E1 -20899.189,E2 -20899.189} C_VEL
LIN {X 0,Y 213.808,Z 512.969,A -85,B 0,C 180,E1 -20903.232,E2 -20903.232} C_VEL
LIN {X 0,Y 213.827,Z 512.945,A -85,B 0,C 180,E1 -20907.451,E2 -20907.451} C_VEL
LIN {X 0,Y 213.768,Z 512.964,A -85,B 0,C 180,E1 -20911.738,E2 -20911.738} C_VEL
LIN {X 0,Y 213.753,Z 512.978,A -85,B 0,C 180,E1 -20916.287,E2 -20916.287} C_VEL
LIN {X 0,Y 213.809,Z 513.104,A -85,B 0,C 180,E1 -20917.92,E2 -20917.92} C_VEL
LIN {X 0,Y 214.427,Z 515.216,A -85,B 0,C 180,E1 -20919.423,E2 -20919.423} C_VEL
LIN {X 0,Y 216.456,Z 518.987,A -85,B 0,C 180,E1 -20920.403,E2 -20920.403} C_VEL
LIN {X 0,Y 218.639,Z 522.187,A -85,B 0,C 180,E1 -20921.222,E2 -20921.222} C_VEL
LIN {X 0,Y 222.331,Z 528.15,A -85,B 0,C 180,E1 -20922.568,E2 -20922.568} C_VEL
LIN {X 0,Y 225.375,Z 533.199,A -85,B 0,C 180,E1 -20923.626,E2 -20923.626} C_VEL
LIN {X 0,Y 230.395,Z 542.065,A -85,B 0,C 180,E1 -20925.293,E2 -20925.293} C_VEL
LIN {X 0,Y 236.925,Z 554.975,A -85,B 0,C 180,E1 -20927.347,E2 -20927.347} C_VEL
LIN {X 0,Y 242.567,Z 567.642,A -85,B 0,C 180,E1 -20929.041,E2 -20929.041} C_VEL
LIN {X 0,Y 245.774,Z 576.06,A -85,B 0,C 180,E1 -20929.997,E2 -20929.997} C_VEL
LIN {X 0,Y 246.953,Z 584.499,A -85,B 0,C 180,E1 -20930.536,E2 -20930.536} C_VEL
LIN {X 0,Y 243.424,Z 652.285,A -85,B 0,C 180,E1 -20932.421,E2 -20932.421} C_VEL
LIN {X 0,Y 243.173,Z 655.664,A -85,B 0,C 180,E1 -20932.544,E2 -20932.544} C_VEL
LIN {X 0,Y 242.082,Z 661.45,A -85,B 0,C 180,E1 -20932.68,E2 -20932.68} C_VEL
LIN {X 0,Y 238.501,Z 670.711,A -85,B 0,C 180,E1 -20932.77,E2 -20932.77} C_VEL
LIN {X 0,Y 234.602,Z 679.815,A -85,B 0,C 180,E1 -20932.986,E2 -20932.986} C_VEL
LIN {X 0,Y 233.002,Z 685.267,A -85,B 0,C 180,E1 -20933.374,E2 -20933.374} C_VEL
LIN {X 0,Y 230.82,Z 695.346,A -85,B 0,C 180,E1 -20934.387,E2 -20934.387} C_VEL
LIN {X 0,Y 228.41,Z 704.974,A -85,B 0,C 180,E1 -20935.572,E2 -20935.572} C_VEL
LIN {X 0,Y 225.705,Z 714.475,A -85,B 0,C 180,E1 -20936.983,E2 -20936.983} C_VEL
LIN {X 0,Y 223.262,Z 722.603,A -85,B 0,C 180,E1 -20938.433,E2 -20938.433} C_VEL
LIN {X 0,Y 220.246,Z 731.669,A -85,B 0,C 180,E1 -20940.357,E2 -20940.357} C_VEL
LIN {X 0,Y 217.668,Z 738.639,A -85,B 0,C 180,E1 -20942.085,E2 -20942.085} C_VEL
LIN {X 0,Y 214.896,Z 746.161,A -85,B 0,C 180,E1 -20944.322,E2 -20944.322} C_VEL
LIN {X 0,Y 211.961,Z 753.773,A -85,B 0,C 180,E1 -20947.071,E2 -20947.071} C_VEL
LIN {X 0,Y 209.926,Z 759.179,A -85,B 0,C 180,E1 -20949.421,E2 -20949.421} C_VEL
LIN {X 0,Y 207.979,Z 764.614,A -85,B 0,C 180,E1 -20952.295,E2 -20952.295} C_VEL
LIN {X 0,Y 206.428,Z 769.063,A -85,B 0,C 180,E1 -20955.206,E2 -20955.206} C_VEL
LIN {X 0,Y 205.34,Z 772.614,A -85,B 0,C 180,E1 -20958.15,E2 -20958.15} C_VEL
LIN {X 0,Y 204.863,Z 774.559,A -85,B 0,C 180,E1 -20960.124,E2 -20960.124} C_VEL
LIN {X 0,Y 204.389,Z 777.255,A -85,B 0,C 180,E1 -20964.079,E2 -20964.079} C_VEL
LIN {X 0,Y 204.343,Z 778.555,A -85,B 0,C 180,E1 -20968.029,E2 -20968.029} C_VEL
LIN {X 0,Y 204.465,Z 778.811,A -85,B 0,C 180,E1 -20970,E2 -20970} C_VEL
LIN {X 0,Y 204.323,Z 778.035,A -85,B 0,C 180,E1 -20974.044,E2 -20974.044} C_VEL
LIN {X 0,Y 204.389,Z 777.255,A -85,B 0,C 180,E1 -20975.921,E2 -20975.921} C_VEL
LIN {X 0,Y 204.863,Z 774.559,A -85,B 0,C 180,E1 -20979.876,E2 -20979.876} C_VEL
LIN {X 0,Y 205.961,Z 770.33,A -85,B 0,C 180,E1 -20983.819,E2 -20983.819} C_VEL
LIN {X 0,Y 207.419,Z 766.195,A -85,B 0,C 180,E1 -20986.738,E2 -20986.738} C_VEL
LIN {X 0,Y 209.201,Z 761.091,A -85,B 0,C 180,E1 -20989.63,E2 -20989.63} C_VEL
LIN {X 0,Y 211.513,Z 754.91,A -85,B 0,C 180,E1 -20992.464,E2 -20992.464} C_VEL
LIN {X 0,Y 213.856,Z 748.836,A -85,B 0,C 180,E1 -20994.771,E2 -20994.771} C_VEL
LIN {X 0,Y 216.469,Z 741.761,A -85,B 0,C 180,E1 -20997.034,E2 -20997.034} C_VEL
LIN {X 0,Y 219.583,Z 733.486,A -85,B 0,C 180,E1 -20999.215,E2 -20999.215} C_VEL
LIN {X 0,Y 222.538,Z 724.921,A -85,B 0,C 180,E1 -21001.102,E2 -21001.102} C_VEL
LIN {X 0,Y 225.268,Z 716.085,A -85,B 0,C 180,E1 -21002.744,E2 -21002.744} C_VEL
LIN {X 0,Y 228.022,Z 706.438,A -85,B 0,C 180,E1 -21004.227,E2 -21004.227} C_VEL
LIN {X 0,Y 230.375,Z 697.098,A -85,B 0,C 180,E1 -21005.423,E2 -21005.423} C_VEL
LIN {X 0,Y 232.745,Z 686.846,A -85,B 0,C 180,E1 -21006.475,E2 -21006.475} C_VEL
LIN {X 0,Y 234.933,Z 675.196,A -85,B 0,C 180,E1 -21007.419,E2 -21007.419} C_VEL
LIN {X 0,Y 236.506,Z 664.672,A -85,B 0,C 180,E1 -21008.068,E2 -21008.068} C_VEL
LIN {X 0,Y 237.746,Z 653.134,A -85,B 0,C 180,E1 -21008.581,E2 -21008.581} C_VEL
LIN {X 0,Y 239.334,Z 626.505,A -85,B 0,C 180,E1 -21009.36,E2 -21009.36} C_VEL
LIN {X 0,Y 241.396,Z 584.185,A -85,B 0,C 180,E1 -21010.563,E2 -21010.563} C_VEL
LIN {X 0,Y 240.249,Z 577.72,A -85,B 0,C 180,E1 -21011.045,E2 -21011.045} C_VEL
LIN {X 0,Y 233.547,Z 561.608,A -85,B 0,C 180,E1 -21013.142,E2 -21013.142} C_VEL
LIN {X 0,Y 226.775,Z 547.783,A -85,B 0,C 180,E1 -21015.361,E2 -21015.361} C_VEL
LIN {X 0,Y 220.31,Z 536.021,A -85,B 0,C 180,E1 -21017.631,E2 -21017.631} C_VEL
LIN {X 0,Y 214.036,Z 525.825,A -85,B 0,C 180,E1 -21020.01,E2 -21020.01} C_VEL
LIN {X 0,Y 211.061,Z 521.105,A -85,B 0,C 180,E1 -21021.225,E2 -21021.225} C_VEL
LIN {X 0,Y 207.515,Z 516.232,A -85,B 0,C 180,E1 -21022.743,E2 -21022.743} C_VEL
LIN {X 0,Y 206.922,Z 514.756,A -85,B 0,C 180,E1 -21023.229,E2 -21023.229} C_VEL
LIN {X 0,Y 206.708,Z 513.91,A -85,B 0,C 180,E1 -21024.092,E2 -21024.092} C_VEL
LIN {X 0,Y 206.718,Z 513.841,A -85,B 0,C 180,E1 -21028.204,E2 -21028.204} C_VEL
LIN {X 0,Y 206.762,Z 513.826,A -85,B 0,C 180,E1 -21032.096,E2 -21032.096} C_VEL
LIN {X 0,Y 206.752,Z 513.85,A -85,B 0,C 180,E1 -21036.603,E2 -21036.603} C_VEL
LIN {X 0,Y 206.87,Z 513.836,A -85,B 0,C 180,E1 -21042.195,E2 -21042.195} C_VEL
LIN {X 0,Y 206.891,Z 513.799,A -85,B 0,C 180,E1 -21046.243,E2 -21046.243} C_VEL
LIN {X 0,Y 207.102,Z 513.813,A -85,B 0,C 180,E1 -21050.23,E2 -21050.23} C_VEL
LIN {X 0,Y 207.163,Z 513.778,A -85,B 0,C 180,E1 -21052.2,E2 -21052.2} C_VEL
LIN {X 0,Y 207.377,Z 513.776,A -85,B 0,C 180,E1 -21058.057,E2 -21058.057} C_VEL
LIN {X 0,Y 207.51,Z 513.733,A -85,B 0,C 180,E1 -21059.999,E2 -21059.999} C_VEL
LIN {X 0,Y 207.376,Z 513.733,A -85,B 0,C 180,E1 -21061.941,E2 -21061.941} C_VEL
LIN {X 0,Y 207.136,Z 513.783,A -85,B 0,C 180,E1 -21067.799,E2 -21067.799} C_VEL
LIN {X 0,Y 206.918,Z 513.807,A -85,B 0,C 180,E1 -21071.758,E2 -21071.758} C_VEL
LIN {X 0,Y 206.858,Z 513.816,A -85,B 0,C 180,E1 -21075.77,E2 -21075.77} C_VEL
LIN {X 0,Y 206.778,Z 513.839,A -85,B 0,C 180,E1 -21079.869,E2 -21079.869} C_VEL
LIN {X 0,Y 206.758,Z 513.822,A -85,B 0,C 180,E1 -21084.072,E2 -21084.072} C_VEL
LIN {X 0,Y 206.739,Z 513.846,A -85,B 0,C 180,E1 -21088.418,E2 -21088.418} C_VEL
LIN {X 0,Y 206.705,Z 513.857,A -85,B 0,C 180,E1 -21092.955,E2 -21092.955} C_VEL
LIN {X 0,Y 206.72,Z 513.994,A -85,B 0,C 180,E1 -21096.811,E2 -21096.811} C_VEL
LIN {X 0,Y 206.891,Z 514.812,A -85,B 0,C 180,E1 -21097.31,E2 -21097.31} C_VEL
LIN {X 0,Y 208.369,Z 517.577,A -85,B 0,C 180,E1 -21098.05,E2 -21098.05} C_VEL
LIN {X 0,Y 210.542,Z 519.628,A -85,B 0,C 180,E1 -21098.914,E2 -21098.914} C_VEL
LIN {X 0,Y 212.682,Z 522.909,A -85,B 0,C 180,E1 -21099.798,E2 -21099.798} C_VEL
LIN {X 0,Y 214.192,Z 524.632,A -85,B 0,C 180,E1 -21100.372,E2 -21100.372} C_VEL
LIN {X 0,Y 216.899,Z 528.268,A -85,B 0,C 180,E1 -21101.391,E2 -21101.391} C_VEL
LIN {X 0,Y 225.19,Z 540.427,A -85,B 0,C 180,E1 -21104.295,E2 -21104.295} C_VEL
LIN {X 0,Y 232.696,Z 552.698,A -85,B 0,C 180,E1 -21106.684,E2 -21106.684} C_VEL
LIN {X 0,Y 244.178,Z 572.9,A -85,B 0,C 180,E1 -21109.958,E2 -21109.958} C_VEL
LIN {X 0,Y 252.221,Z 584.119,A -85,B 0,C 180,E1 -21111.887,E2 -21111.887} C_VEL
LIN {X 0,Y 263.768,Z 597.475,A -85,B 0,C 180,E1 -21114.283,E2 -21114.283} C_VEL
LIN {X 0,Y 281.488,Z 614.383,A -85,B 0,C 180,E1 -21117.359,E2 -21117.359} C_VEL
LIN {X 0,Y 292.635,Z 623.671,A -85,B 0,C 180,E1 -21119.072,E2 -21119.072} C_VEL
LIN {X 0,Y 301.827,Z 631.102,A -85,B 0,C 180,E1 -21120.644,E2 -21120.644} C_VEL
LIN {X 0,Y 309.883,Z 637.388,A -85,B 0,C 180,E1 -21122.189,E2 -21122.189} C_VEL
LIN {X 0,Y 318.665,Z 644.125,A -85,B 0,C 180,E1 -21124.124,E2 -21124.124} C_VEL
LIN {X 0,Y 326.289,Z 649.833,A -85,B 0,C 180,E1 -21125.981,E2 -21125.981} C_VEL
LIN {X 0,Y 333.471,Z 655.183,A -85,B 0,C 180,E1 -21127.892,E2 -21127.892} C_VEL
LIN {X 0,Y 340.405,Z 659.939,A -85,B 0,C 180,E1 -21129.898,E2 -21129.898} C_VEL
LIN {X 0,Y 346.969,Z 664.75,A -85,B 0,C 180,E1 -21132.038,E2 -21132.038} C_VEL
LIN {X 0,Y 352.355,Z 668.361,A -85,B 0,C 180,E1 -21134.013,E2 -21134.013} C_VEL
LIN {X 0,Y 357.498,Z 671.31,A -85,B 0,C 180,E1 -21136.112,E2 -21136.112} C_VEL
LIN {X 0,Y 361.634,Z 674.559,A -85,B 0,C 180,E1 -21138.151,E2 -21138.151} C_VEL
LIN {X 0,Y 365.398,Z 676.965,A -85,B 0,C 180,E1 -21140.331,E2 -21140.331} C_VEL
LIN {X 0,Y 368.542,Z 678.621,A -85,B 0,C 180,E1 -21142.574,E2 -21142.574} C_VEL
LIN {X 0,Y 370.662,Z 679.614,A -85,B 0,C 180,E1 -21144.56,E2 -21144.56} C_VEL
LIN {X 0,Y 372.314,Z 680.145,A -85,B 0,C 180,E1 -21146.754,E2 -21146.754} C_VEL
LIN {X 0,Y 373.071,Z 680.571,A -85,B 0,C 180,E1 -21148.921,E2 -21148.921} C_VEL
LIN {X 0,Y 373.197,Z 680.469,A -85,B 0,C 180,E1 -21150,E2 -21150} C_VEL
LIN {X 0,Y 373.052,Z 680.588,A -85,B 0,C 180,E1 -21151.079,E2 -21151.079} C_VEL
LIN {X 0,Y 372.303,Z 680.145,A -85,B 0,C 180,E1 -21153.246,E2 -21153.246} C_VEL
LIN {X 0,Y 370.674,Z 679.627,A -85,B 0,C 180,E1 -21155.44,E2 -21155.44} C_VEL
LIN {X 0,Y 368.203,Z 678.497,A -85,B 0,C 180,E1 -21157.678,E2 -21157.678} C_VEL
LIN {X 0,Y 365.221,Z 676.824,A -85,B 0,C 180,E1 -21159.791,E2 -21159.791} C_VEL
LIN {X 0,Y 361.293,Z 674.331,A -85,B 0,C 180,E1 -21162.017,E2 -21162.017} C_VEL
LIN {X 0,Y 356.937,Z 670.859,A -85,B 0,C 180,E1 -21164.148,E2 -21164.148} C_VEL
LIN {X 0,Y 351.176,Z 667.637,A -85,B 0,C 180,E1 -21166.424,E2 -21166.424} C_VEL
LIN {X 0,Y 346.252,Z 664.266,A -85,B 0,C 180,E1 -21168.183,E2 -21168.183} C_VEL
LIN {X 0,Y 339.967,Z 659.626,A -85,B 0,C 180,E1 -21170.233,E2 -21170.233} C_VEL
LIN {X 0,Y 333.934,Z 655.563,A -85,B 0,C 180,E1 -21171.974,E2 -21171.974} C_VEL
LIN {X 0,Y 326.804,Z 650.182,A -85,B 0,C 180,E1 -21173.885,E2 -21173.885} C_VEL
LIN {X 0,Y 319.63,Z 644.887,A -85,B 0,C 180,E1 -21175.645,E2 -21175.645} C_VEL
LIN {X 0,Y 312.169,Z 639.15,A -85,B 0,C 180,E1 -21177.329,E2 -21177.329} C_VEL
LIN {X 0,Y 305.258,Z 633.613,A -85,B 0,C 180,E1 -21178.727,E2 -21178.727} C_VEL
LIN {X 0,Y 297.538,Z 627.725,A -85,B 0,C 180,E1 -21180.107,E2 -21180.107} C_VEL
LIN {X 0,Y 289.502,Z 621.195,A -85,B 0,C 180,E1 -21181.412,E2 -21181.412} C_VEL
LIN {X 0,Y 274.972,Z 608.426,A -85,B 0,C 180,E1 -21183.705,E2 -21183.705} C_VEL
LIN {X 0,Y 260.99,Z 594.403,A -85,B 0,C 180,E1 -21186.262,E2 -21186.262} C_VEL
LIN {X 0,Y 250.403,Z 581.852,A -85,B 0,C 180,E1 -21188.524,E2 -21188.524} C_VEL
LIN {X 0,Y 241.77,Z 568.981,A -85,B 0,C 180,E1 -21190.677,E2 -21190.677} C_VEL
LIN {X 0,Y 231.048,Z 549.861,A -85,B 0,C 180,E1 -21193.825,E2 -21193.825} C_VEL
LIN {X 0,Y 223.436,Z 537.816,A -85,B 0,C 180,E1 -21196.291,E2 -21196.291} C_VEL
LIN {X 0,Y 218.686,Z 531.006,A -85,B 0,C 180,E1 -21197.945,E2 -21197.945} C_VEL
LIN {X 0,Y 216.24,Z 527.589,A -85,B 0,C 180,E1 -21198.843,E2 -21198.843} C_VEL
LIN {X 0,Y 213.335,Z 523.553,A -85,B 0,C 180,E1 -21199.957,E2 -21199.957} C_VEL
LIN {X 0,Y 211.048,Z 520.609,A -85,B 0,C 180,E1 -21200.863,E2 -21200.863} C_VEL
LIN {X 0,Y 210.035,Z 519.016,A -85,B 0,C 180,E1 -21201.292,E2 -21201.292} C_VEL
LIN {X 0,Y 207.846,Z 516.884,A -85,B 0,C 180,E1 -21202.174,E2 -21202.174} C_VEL
LIN {X 0,Y 206.856,Z 514.606,A -85,B 0,C 180,E1 -21202.76,E2 -21202.76} C_VEL
LIN {X 0,Y 206.716,Z 513.914,A -85,B 0,C 180,E1 -21203.34,E2 -21203.34} C_VEL
LIN {X 0,Y 206.724,Z 513.838,A -85,B 0,C 180,E1 -21208.201,E2 -21208.201} C_VEL
LIN {X 0,Y 206.762,Z 513.853,A -85,B 0,C 180,E1 -21212.097,E2 -21212.097} C_VEL
LIN {X 0,Y 206.78,Z 513.822,A -85,B 0,C 180,E1 -21216.585,E2 -21216.585} C_VEL
LIN {X 0,Y 206.868,Z 513.805,A -85,B 0,C 180,E1 -21222.197,E2 -21222.197} C_VEL
LIN {X 0,Y 206.888,Z 513.841,A -85,B 0,C 180,E1 -21226.245,E2 -21226.245} C_VEL
LIN {X 0,Y 207.095,Z 513.771,A -85,B 0,C 180,E1 -21230.232,E2 -21230.232} C_VEL
LIN {X 0,Y 207.058,Z 513.816,A -85,B 0,C 180,E1 -21234.157,E2 -21234.157} C_VEL
LIN {X 0,Y 207.377,Z 513.732,A -85,B 0,C 180,E1 -21238.059,E2 -21238.059} C_VEL
LIN {X 0,Y 207.51,Z 513.733,A -85,B 0,C 180,E1 -21240.001,E2 -21240.001} C_VEL
LIN {X 0,Y 207.377,Z 513.776,A -85,B 0,C 180,E1 -21241.943,E2 -21241.943} C_VEL
LIN {X 0,Y 207.163,Z 513.778,A -85,B 0,C 180,E1 -21247.8,E2 -21247.8} C_VEL
LIN {X 0,Y 206.939,Z 513.804,A -85,B 0,C 180,E1 -21251.758,E2 -21251.758} C_VEL
LIN {X 0,Y 206.862,Z 513.823,A -85,B 0,C 180,E1 -21255.772,E2 -21255.772} C_VEL
LIN {X 0,Y 206.759,Z 513.822,A -85,B 0,C 180,E1 -21259.872,E2 -21259.872} C_VEL
LIN {X 0,Y 206.744,Z 513.858,A -85,B 0,C 180,E1 -21264.075,E2 -21264.075} C_VEL
LIN {X 0,Y 206.735,Z 513.833,A -85,B 0,C 180,E1 -21268.421,E2 -21268.421} C_VEL
LIN {X 0,Y 206.704,Z 513.836,A -85,B 0,C 180,E1 -21272.958,E2 -21272.958} C_VEL
LIN {X 0,Y 206.739,Z 514.002,A -85,B 0,C 180,E1 -21276.203,E2 -21276.203} C_VEL
LIN {X 0,Y 207.135,Z 515.397,A -85,B 0,C 180,E1 -21277.032,E2 -21277.032} C_VEL
LIN {X 0,Y 210.12,Z 519.941,A -85,B 0,C 180,E1 -21278.395,E2 -21278.395} C_VEL
LIN {X 0,Y 211.376,Z 521.734,A -85,B 0,C 180,E1 -21278.914,E2 -21278.914} C_VEL
LIN {X 0,Y 215.852,Z 528.856,A -85,B 0,C 180,E1 -21280.709,E2 -21280.709} C_VEL
LIN {X 0,Y 218.634,Z 533.354,A -85,B 0,C 180,E1 -21281.76,E2 -21281.76} C_VEL
LIN {X 0,Y 223.796,Z 542.216,A -85,B 0,C 180,E1 -21283.614,E2 -21283.614} C_VEL
LIN {X 0,Y 229.909,Z 553.919,A -85,B 0,C 180,E1 -21285.681,E2 -21285.681} C_VEL
LIN {X 0,Y 236.326,Z 567.95,A -85,B 0,C 180,E1 -21287.736,E2 -21287.736} C_VEL
LIN {X 0,Y 240.509,Z 578.615,A -85,B 0,C 180,E1 -21289.043,E2 -21289.043} C_VEL
LIN {X 0,Y 241.46,Z 585.405,A -85,B 0,C 180,E1 -21289.497,E2 -21289.497} C_VEL
LIN {X 0,Y 237.819,Z 652.414,A -85,B 0,C 180,E1 -21291.391,E2 -21291.391} C_VEL
LIN {X 0,Y 236.498,Z 664.672,A -85,B 0,C 180,E1 -21291.931,E2 -21291.931} C_VEL
LIN {X 0,Y 234.484,Z 677.915,A -85,B 0,C 180,E1 -21292.768,E2 -21292.768} C_VEL
LIN {X 0,Y 233.002,Z 685.267,A -85,B 0,C 180,E1 -21293.374,E2 -21293.374} C_VEL
LIN {X 0,Y 231.332,Z 690.826,A -85,B 0,C 180,E1 -21293.789,E2 -21293.789} C_VEL
LIN {X 0,Y 226.908,Z 699.363,A -85,B 0,C 180,E1 -21294.312,E2 -21294.312} C_VEL
LIN {X 0,Y 222.26,Z 707.687,A -85,B 0,C 180,E1 -21295.003,E2 -21295.003} C_VEL
LIN {X 0,Y 220.265,Z 712.578,A -85,B 0,C 180,E1 -21295.681,E2 -21295.681} C_VEL
LIN {X 0,Y 217.436,Z 721.767,A -85,B 0,C 180,E1 -21297.32,E2 -21297.32} C_VEL
LIN {X 0,Y 214.093,Z 731.47,A -85,B 0,C 180,E1 -21299.416,E2 -21299.416} C_VEL
LIN {X 0,Y 211.408,Z 738.44,A -85,B 0,C 180,E1 -21301.182,E2 -21301.182} C_VEL
LIN {X 0,Y 208.495,Z 745.963,A -85,B 0,C 180,E1 -21303.473,E2 -21303.473} C_VEL
LIN {X 0,Y 205.386,Z 753.573,A -85,B 0,C 180,E1 -21306.293,E2 -21306.293} C_VEL
LIN {X 0,Y 203.232,Z 758.979,A -85,B 0,C 180,E1 -21308.711,E2 -21308.711} C_VEL
LIN {X 0,Y 201.181,Z 764.415,A -85,B 0,C 180,E1 -21311.676,E2 -21311.676} C_VEL
LIN {X 0,Y 199.536,Z 768.864,A -85,B 0,C 180,E1 -21314.683,E2 -21314.683} C_VEL
LIN {X 0,Y 198.346,Z 772.414,A -85,B 0,C 180,E1 -21317.726,E2 -21317.726} C_VEL
LIN {X 0,Y 197.848,Z 774.36,A -85,B 0,C 180,E1 -21319.77,E2 -21319.77} C_VEL
LIN {X 0,Y 197.304,Z 777.056,A -85,B 0,C 180,E1 -21323.866,E2 -21323.866} C_VEL
LIN {X 0,Y 197.248,Z 777.946,A -85,B 0,C 180,E1 -21326.081,E2 -21326.081} C_VEL
LIN {X 0,Y 197.365,Z 778.613,A -85,B 0,C 180,E1 -21330,E2 -21330} C_VEL
LIN {X 0,Y 197.248,Z 777.879,A -85,B 0,C 180,E1 -21334.086,E2 -21334.086} C_VEL
LIN {X 0,Y 197.304,Z 777.056,A -85,B 0,C 180,E1 -21336.134,E2 -21336.134} C_VEL
LIN {X 0,Y 197.848,Z 774.36,A -85,B 0,C 180,E1 -21340.23,E2 -21340.23} C_VEL
LIN {X 0,Y 199.032,Z 770.131,A -85,B 0,C 180,E1 -21344.31,E2 -21344.31} C_VEL
LIN {X 0,Y 200.563,Z 765.995,A -85,B 0,C 180,E1 -21347.328,E2 -21347.328} C_VEL
LIN {X 0,Y 201.834,Z 762.798,A -85,B 0,C 180,E1 -21349.317,E2 -21349.317} C_VEL
LIN {X 0,Y 204.473,Z 755.849,A -85,B 0,C 180,E1 -21352.747,E2 -21352.747} C_VEL
LIN {X 0,Y 207.395,Z 748.637,A -85,B 0,C 180,E1 -21355.598,E2 -21355.598} C_VEL
LIN {X 0,Y 210.133,Z 741.562,A -85,B 0,C 180,E1 -21357.919,E2 -21357.919} C_VEL
LIN {X 0,Y 213.402,Z 733.288,A -85,B 0,C 180,E1 -21360.147,E2 -21360.147} C_VEL
LIN {X 0,Y 216.699,Z 724.086,A -85,B 0,C 180,E1 -21362.203,E2 -21362.203} C_VEL
LIN {X 0,Y 219.404,Z 715.512,A -85,B 0,C 180,E1 -21363.817,E2 -21363.817} C_VEL
LIN {X 0,Y 222.179,Z 706.24,A -85,B 0,C 180,E1 -21365.259,E2 -21365.259} C_VEL
LIN {X 0,Y 224.618,Z 696.9,A -85,B 0,C 180,E1 -21366.475,E2 -21366.475} C_VEL
LIN {X 0,Y 227.058,Z 686.647,A -85,B 0,C 180,E1 -21367.543,E2 -21367.543} C_VEL
LIN {X 0,Y 229.344,Z 674.998,A -85,B 0,C 180,E1 -21368.495,E2 -21368.495} C_VEL
LIN {X 0,Y 231.076,Z 663.562,A -85,B 0,C 180,E1 -21369.2,E2 -21369.2} C_VEL
LIN {X 0,Y 232.279,Z 652.432,A -85,B 0,C 180,E1 -21369.691,E2 -21369.691} C_VEL
LIN {X 0,Y 234.021,Z 623.651,A -85,B 0,C 180,E1 -21370.541,E2 -21370.541} C_VEL
LIN {X 0,Y 236.005,Z 585.437,A -85,B 0,C 180,E1 -21371.635,E2 -21371.635} C_VEL
LIN {X 0,Y 235.105,Z 580.613,A -85,B 0,C 180,E1 -21372.022,E2 -21372.022} C_VEL
LIN {X 0,Y 228.898,Z 565.499,A -85,B 0,C 180,E1 -21374.069,E2 -21374.069} C_VEL
LIN {X 0,Y 222.467,Z 552.142,A -85,B 0,C 180,E1 -21376.289,E2 -21376.289} C_VEL
LIN {X 0,Y 216.475,Z 541.015,A -85,B 0,C 180,E1 -21378.503,E2 -21378.503} C_VEL
LIN {X 0,Y 212.655,Z 534.701,A -85,B 0,C 180,E1 -21379.995,E2 -21379.995} C_VEL
LIN {X 0,Y 209.814,Z 530.086,A -85,B 0,C 180,E1 -21381.167,E2 -21381.167} C_VEL
LIN {X 0,Y 206.726,Z 525.314,A -85,B 0,C 180,E1 -21382.5,E2 -21382.5} C_VEL
LIN {X 0,Y 203.023,Z 519.941,A -85,B 0,C 180,E1 -21384.189,E2 -21384.189} C_VEL
LIN {X 0,Y 200.665,Z 517.601,A -85,B 0,C 180,E1 -21385.269,E2 -21385.269} C_VEL
LIN {X 0,Y 199.733,Z 515.268,A -85,B 0,C 180,E1 -21386.002,E2 -21386.002} C_VEL
LIN {X 0,Y 199.673,Z 514.739,A -85,B 0,C 180,E1 -21386.784,E2 -21386.784} C_VEL
LIN {X 0,Y 199.706,Z 514.708,A -85,B 0,C 180,E1 -21391.615,E2 -21391.615} C_VEL
LIN {X 0,Y 199.711,Z 514.714,A -85,B 0,C 180,E1 -21397.225,E2 -21397.225} C_VEL
LIN {X 0,Y 199.793,Z 514.708,A -85,B 0,C 180,E1 -21401.758,E2 -21401.758} C_VEL
LIN {X 0,Y 199.831,Z 514.68,A -85,B 0,C 180,E1 -21405.747,E2 -21405.747} C_VEL
LIN {X 0,Y 200.067,Z 514.687,A -85,B 0,C 180,E1 -21409.883,E2 -21409.883} C_VEL
LIN {X 0,Y 200.029,Z 514.649,A -85,B 0,C 180,E1 -21413.949,E2 -21413.949} C_VEL
LIN {X 0,Y 200.317,Z 514.655,A -85,B 0,C 180,E1 -21417.988,E2 -21417.988} C_VEL
LIN {X 0,Y 200.474,Z 514.608,A -85,B 0,C 180,E1 -21419.999,E2 -21419.999} C_VEL
LIN {X 0,Y 200.021,Z 514.662,A -85,B 0,C 180,E1 -21424.029,E2 -21424.029} C_VEL
LIN {X 0,Y 200.084,Z 514.656,A -85,B 0,C 180,E1 -21428.076,E2 -21428.076} C_VEL
LIN {X 0,Y 199.868,Z 514.691,A -85,B 0,C 180,E1 -21432.179,E2 -21432.179} C_VEL
LIN {X 0,Y 199.797,Z 514.688,A -85,B 0,C 180,E1 -21436.343,E2 -21436.343} C_VEL
LIN {X 0,Y 199.695,Z 514.734,A -85,B 0,C 180,E1 -21440.605,E2 -21440.605} C_VEL
LIN {X 0,Y 199.668,Z 514.706,A -85,B 0,C 180,E1 -21444.984,E2 -21444.984} C_VEL
LIN {X 0,Y 199.67,Z 514.713,A -85,B 0,C 180,E1 -21449.522,E2 -21449.522} C_VEL
LIN {X 0,Y 199.639,Z 514.792,A -85,B 0,C 180,E1 -21453.948,E2 -21453.948} C_VEL
LIN {X 0,Y 199.842,Z 515.725,A -85,B 0,C 180,E1 -21454.612,E2 -21454.612} C_VEL
LIN {X 0,Y 201.398,Z 518.552,A -85,B 0,C 180,E1 -21455.478,E2 -21455.478} C_VEL
LIN {X 0,Y 203.618,Z 520.448,A -85,B 0,C 180,E1 -21456.463,E2 -21456.463} C_VEL
LIN {X 0,Y 205.659,Z 523.742,A -85,B 0,C 180,E1 -21457.418,E2 -21457.418} C_VEL
LIN {X 0,Y 207.446,Z 525.598,A -85,B 0,C 180,E1 -21458.165,E2 -21458.165} C_VEL
LIN {X 0,Y 210.145,Z 529.312,A -85,B 0,C 180,E1 -21459.296,E2 -21459.296} C_VEL
LIN {X 0,Y 214.949,Z 536.11,A -85,B 0,C 180,E1 -21461.186,E2 -21461.186} C_VEL
LIN {X 0,Y 221.225,Z 545.292,A -85,B 0,C 180,E1 -21463.451,E2 -21463.451} C_VEL
LIN {X 0,Y 229.575,Z 559.283,A -85,B 0,C 180,E1 -21466.221,E2 -21466.221} C_VEL
LIN {X 0,Y 239.325,Z 576.892,A -85,B 0,C 180,E1 -21469.123,E2 -21469.123} C_VEL
LIN {X 0,Y 247.599,Z 588.701,A -85,B 0,C 180,E1 -21471.204,E2 -21471.204} C_VEL
LIN {X 0,Y 259.093,Z 602.255,A -85,B 0,C 180,E1 -21473.693,E2 -21473.693} C_VEL
LIN {X 0,Y 276.867,Z 619.442,A -85,B 0,C 180,E1 -21476.894,E2 -21476.894} C_VEL
LIN {X 0,Y 289.307,Z 629.808,A -85,B 0,C 180,E1 -21478.819,E2 -21478.819} C_VEL
LIN {X 0,Y 297.695,Z 636.519,A -85,B 0,C 180,E1 -21480.179,E2 -21480.179} C_VEL
LIN {X 0,Y 305.742,Z 642.751,A -85,B 0,C 180,E1 -21481.68,E2 -21481.68} C_VEL
LIN {X 0,Y 313.6,Z 648.603,A -85,B 0,C 180,E1 -21483.335,E2 -21483.335} C_VEL
LIN {X 0,Y 320.815,Z 654.253,A -85,B 0,C 180,E1 -21485.033,E2 -21485.033} C_VEL
LIN {X 0,Y 327.804,Z 659.265,A -85,B 0,C 180,E1 -21486.794,E2 -21486.794} C_VEL
LIN {X 0,Y 334.601,Z 664.231,A -85,B 0,C 180,E1 -21488.678,E2 -21488.678} C_VEL
LIN {X 0,Y 340.774,Z 668.411,A -85,B 0,C 180,E1 -21490.548,E2 -21490.548} C_VEL
LIN {X 0,Y 346.397,Z 672.638,A -85,B 0,C 180,E1 -21492.471,E2 -21492.471} C_VEL
LIN {X 0,Y 351.744,Z 675.923,A -85,B 0,C 180,E1 -21494.443,E2 -21494.443} C_VEL
LIN {X 0,Y 355.919,Z 678.408,A -85,B 0,C 180,E1 -21496.188,E2 -21496.188} C_VEL
LIN {X 0,Y 360.02,Z 681.627,A -85,B 0,C 180,E1 -21498.264,E2 -21498.264} C_VEL
LIN {X 0,Y 363.583,Z 683.856,A -85,B 0,C 180,E1 -21500.335,E2 -21500.335} C_VEL
LIN {X 0,Y 366.377,Z 685.293,A -85,B 0,C 180,E1 -21502.283,E2 -21502.283} C_VEL
LIN {X 0,Y 368.85,Z 686.475,A -85,B 0,C 180,E1 -21504.533,E2 -21504.533} C_VEL
LIN {X 0,Y 370.523,Z 687.015,A -85,B 0,C 180,E1 -21506.738,E2 -21506.738} C_VEL
LIN {X 0,Y 371.274,Z 687.426,A -85,B 0,C 180,E1 -21508.915,E2 -21508.915} C_VEL
LIN {X 0,Y 371.401,Z 687.339,A -85,B 0,C 180,E1 -21510,E2 -21510} C_VEL
LIN {X 0,Y 371.256,Z 687.456,A -85,B 0,C 180,E1 -21511.085,E2 -21511.085} C_VEL
LIN {X 0,Y 370.5,Z 687.012,A -85,B 0,C 180,E1 -21513.262,E2 -21513.262} C_VEL
LIN {X 0,Y 368.865,Z 686.478,A -85,B 0,C 180,E1 -21515.466,E2 -21515.466} C_VEL
LIN {X 0,Y 366.368,Z 685.326,A -85,B 0,C 180,E1 -21517.717,E2 -21517.717} C_VEL
LIN {X 0,Y 363.012,Z 683.461,A -85,B 0,C 180,E1 -21520.034,E2 -21520.034} C_VEL
LIN {X 0,Y 359.018,Z 680.871,A -85,B 0,C 180,E1 -21522.265,E2 -21522.265} C_VEL
LIN {X 0,Y 354.515,Z 677.379,A -85,B 0,C 180,E1 -21524.44,E2 -21524.44} C_VEL
LIN {X 0,Y 348.493,Z 673.974,A -85,B 0,C 180,E1 -21526.781,E2 -21526.781} C_VEL
LIN {X 0,Y 343.19,Z 670.339,A -85,B 0,C 180,E1 -21528.626,E2 -21528.626} C_VEL
LIN {X 0,Y 337.805,Z 666.344,A -85,B 0,C 180,E1 -21530.37,E2 -21530.37} C_VEL
LIN {X 0,Y 331.057,Z 661.778,A -85,B 0,C 180,E1 -21532.313,E2 -21532.313} C_VEL
LIN {X 0,Y 323.748,Z 656.322,A -85,B 0,C 180,E1 -21534.254,E2 -21534.254} C_VEL
LIN {X 0,Y 315.979,Z 650.553,A -85,B 0,C 180,E1 -21536.119,E2 -21536.119} C_VEL
LIN {X 0,Y 307.005,Z 643.738,A -85,B 0,C 180,E1 -21538.065,E2 -21538.065} C_VEL
LIN {X 0,Y 299.039,Z 637.496,A -85,B 0,C 180,E1 -21539.593,E2 -21539.593} C_VEL
LIN {X 0,Y 290.878,Z 631.04,A -85,B 0,C 180,E1 -21540.939,E2 -21540.939} C_VEL
LIN {X 0,Y 280.1,Z 622.198,A -85,B 0,C 180,E1 -21542.591,E2 -21542.591} C_VEL
LIN {X 0,Y 265.95,Z 609.206,A -85,B 0,C 180,E1 -21544.996,E2 -21544.996} C_VEL
LIN {X 0,Y 253.95,Z 596.468,A -85,B 0,C 180,E1 -21547.373,E2 -21547.373} C_VEL
LIN {X 0,Y 243.54,Z 583.252,A -85,B 0,C 180,E1 -21549.778,E2 -21549.778} C_VEL
LIN {X 0,Y 235.716,Z 570.75,A -85,B 0,C 180,E1 -21551.892,E2 -21551.892} C_VEL
LIN {X 0,Y 226.926,Z 554.651,A -85,B 0,C 180,E1 -21554.63,E2 -21554.63} C_VEL
LIN {X 0,Y 219.564,Z 542.811,A -85,B 0,C 180,E1 -21557.129,E2 -21557.129} C_VEL
LIN {X 0,Y 213.053,Z 533.339,A -85,B 0,C 180,E1 -21559.546,E2 -21559.546} C_VEL
LIN {X 0,Y 209.769,Z 528.914,A -85,B 0,C 180,E1 -21560.852,E2 -21560.852} C_VEL
LIN {X 0,Y 206.784,Z 524.809,A -85,B 0,C 180,E1 -21562.115,E2 -21562.115} C_VEL
LIN {X 0,Y 204.381,Z 521.968,A -85,B 0,C 180,E1 -21563.159,E2 -21563.159} C_VEL
LIN {X 0,Y 203.264,Z 520.091,A -85,B 0,C 180,E1 -21563.694,E2 -21563.694} C_VEL
LIN {X 0,Y 200.971,Z 517.989,A -85,B 0,C 180,E1 -21564.728,E2 -21564.728} C_VEL
LIN {X 0,Y 199.759,Z 515.302,A -85,B 0,C 180,E1 -21565.558,E2 -21565.558} C_VEL
LIN {X 0,Y 199.661,Z 514.766,A -85,B 0,C 180,E1 -21566.255,E2 -21566.255} C_VEL
LIN {X 0,Y 199.67,Z 514.713,A -85,B 0,C 180,E1 -21570.478,E2 -21570.478} C_VEL
LIN {X 0,Y 199.668,Z 514.706,A -85,B 0,C 180,E1 -21575.016,E2 -21575.016} C_VEL
LIN {X 0,Y 199.695,Z 514.734,A -85,B 0,C 180,E1 -21579.395,E2 -21579.395} C_VEL
LIN {X 0,Y 199.797,Z 514.688,A -85,B 0,C 180,E1 -21583.657,E2 -21583.657} C_VEL
LIN {X 0,Y 199.868,Z 514.691,A -85,B 0,C 180,E1 -21587.821,E2 -21587.821} C_VEL
LIN {X 0,Y 200.084,Z 514.656,A -85,B 0,C 180,E1 -21591.924,E2 -21591.924} C_VEL
LIN {X 0,Y 200.317,Z 514.611,A -85,B 0,C 180,E1 -21597.99,E2 -21597.99} C_VEL
LIN {X 0,Y 200.475,Z 514.608,A -85,B 0,C 180,E1 -21600.001,E2 -21600.001} C_VEL
LIN {X 0,Y 200.024,Z 514.66,A -85,B 0,C 180,E1 -21604.031,E2 -21604.031} C_VEL
LIN {X 0,Y 200.107,Z 514.66,A -85,B 0,C 180,E1 -21608.077,E2 -21608.077} C_VEL
LIN {X 0,Y 200.033,Z 514.689,A -85,B 0,C 180,E1 -21610.348,E2 -21610.348} C_VEL
LIN {X 0,Y 199.831,Z 514.68,A -85,B 0,C 180,E1 -21614.253,E2 -21614.253} C_VEL
LIN {X 0,Y 199.778,Z 514.707,A -85,B 0,C 180,E1 -21618.459,E2 -21618.459} C_VEL
LIN {X 0,Y 199.712,Z 514.732,A -85,B 0,C 180,E1 -21623.804,E2 -21623.804} C_VEL
LIN {X 0,Y 199.706,Z 514.708,A -85,B 0,C 180,E1 -21628.385,E2 -21628.385} C_VEL
LIN {X 0,Y 199.673,Z 514.735,A -85,B 0,C 180,E1 -21633.216,E2 -21633.216} C_VEL
LIN {X 0,Y 199.726,Z 515.277,A -85,B 0,C 180,E1 -21633.999,E2 -21633.999} C_VEL
LIN {X 0,Y 200.798,Z 517.802,A -85,B 0,C 180,E1 -21634.797,E2 -21634.797} C_VEL
LIN {X 0,Y 203.846,Z 520.962,A -85,B 0,C 180,E1 -21636.188,E2 -21636.188} C_VEL
LIN {X 0,Y 208.103,Z 527.398,A -85,B 0,C 180,E1 -21638.102,E2 -21638.102} C_VEL
LIN {X 0,Y 212.294,Z 534.095,A -85,B 0,C 180,E1 -21639.858,E2 -21639.858} C_VEL
LIN {X 0,Y 217.04,Z 542.096,A -85,B 0,C 180,E1 -21641.716,E2 -21641.716} C_VEL
LIN {X 0,Y 223.395,Z 553.826,A -85,B 0,C 180,E1 -21644.034,E2 -21644.034} C_VEL
LIN {X 0,Y 230.121,Z 568.258,A -85,B 0,C 180,E1 -21646.339,E2 -21646.339} C_VEL
LIN {X 0,Y 235.347,Z 581.291,A -85,B 0,C 180,E1 -21648.058,E2 -21648.058} C_VEL
LIN {X 0,Y 236.061,Z 586.438,A -85,B 0,C 180,E1 -21648.417,E2 -21648.417} C_VEL
LIN {X 0,Y 232.371,Z 651.787,A -85,B 0,C 180,E1 -21650.287,E2 -21650.287} C_VEL
LIN {X 0,Y 231.079,Z 663.562,A -85,B 0,C 180,E1 -21650.801,E2 -21650.801} C_VEL
LIN {X 0,Y 229.335,Z 674.998,A -85,B 0,C 180,E1 -21651.504,E2 -21651.504} C_VEL
LIN {X 0,Y 227.033,Z 686.646,A -85,B 0,C 180,E1 -21652.452,E2 -21652.452} C_VEL
LIN {X 0,Y 223.794,Z 700.356,A -85,B 0,C 180,E1 -21653.928,E2 -21653.928} C_VEL
LIN {X 0,Y 220.265,Z 712.578,A -85,B 0,C 180,E1 -21655.681,E2 -21655.681} C_VEL
LIN {X 0,Y 218.241,Z 717.552,A -85,B 0,C 180,E1 -21656.427,E2 -21656.427} C_VEL
LIN {X 0,Y 213.257,Z 725.09,A -85,B 0,C 180,E1 -21657.505,E2 -21657.505} C_VEL
LIN {X 0,Y 208.172,Z 732.218,A -85,B 0,C 180,E1 -21658.73,E2 -21658.73} C_VEL
LIN {X 0,Y 205.998,Z 736.381,A -85,B 0,C 180,E1 -21659.694,E2 -21659.694} C_VEL
LIN {X 0,Y 202.111,Z 745.763,A -85,B 0,C 180,E1 -21662.566,E2 -21662.566} C_VEL
LIN {X 0,Y 199.379,Z 752.236,A -85,B 0,C 180,E1 -21664.977,E2 -21664.977} C_VEL
LIN {X 0,Y 196.576,Z 758.777,A -85,B 0,C 180,E1 -21667.952,E2 -21667.952} C_VEL
LIN {X 0,Y 194.409,Z 764.216,A -85,B 0,C 180,E1 -21671.013,E2 -21671.013} C_VEL
LIN {X 0,Y 192.666,Z 768.665,A -85,B 0,C 180,E1 -21674.123,E2 -21674.123} C_VEL
LIN {X 0,Y 191.348,Z 772.214,A -85,B 0,C 180,E1 -21677.269,E2 -21677.269} C_VEL
LIN {X 0,Y 190.818,Z 774.161,A -85,B 0,C 180,E1 -21679.388,E2 -21679.388} C_VEL
LIN {X 0,Y 190.221,Z 776.857,A -85,B 0,C 180,E1 -21683.636,E2 -21683.636} C_VEL
LIN {X 0,Y 190.156,Z 777.887,A -85,B 0,C 180,E1 -21686.294,E2 -21686.294} C_VEL
LIN {X 0,Y 190.267,Z 778.415,A -85,B 0,C 180,E1 -21690,E2 -21690} C_VEL
LIN {X 0,Y 190.164,Z 777.681,A -85,B 0,C 180,E1 -21694.239,E2 -21694.239} C_VEL
LIN {X 0,Y 190.221,Z 776.857,A -85,B 0,C 180,E1 -21696.364,E2 -21696.364} C_VEL
LIN {X 0,Y 190.818,Z 774.161,A -85,B 0,C 180,E1 -21700.612,E2 -21700.612} C_VEL
LIN {X 0,Y 192.126,Z 769.932,A -85,B 0,C 180,E1 -21704.836,E2 -21704.836} C_VEL
LIN {X 0,Y 193.735,Z 765.795,A -85,B 0,C 180,E1 -21707.959,E2 -21707.959} C_VEL
LIN {X 0,Y 195.742,Z 760.691,A -85,B 0,C 180,E1 -21711.041,E2 -21711.041} C_VEL
LIN {X 0,Y 198.376,Z 754.512,A -85,B 0,C 180,E1 -21714.042,E2 -21714.042} C_VEL
LIN {X 0,Y 200.971,Z 748.438,A -85,B 0,C 180,E1 -21716.478,E2 -21716.478} C_VEL
LIN {X 0,Y 203.851,Z 741.362,A -85,B 0,C 180,E1 -21718.859,E2 -21718.859} C_VEL
LIN {X 0,Y 207.285,Z 733.089,A -85,B 0,C 180,E1 -21721.134,E2 -21721.134} C_VEL
LIN {X 0,Y 210.559,Z 724.292,A -85,B 0,C 180,E1 -21723.152,E2 -21723.152} C_VEL
LIN {X 0,Y 213.526,Z 715.314,A -85,B 0,C 180,E1 -21724.88,E2 -21724.88} C_VEL
LIN {X 0,Y 216.392,Z 706.041,A -85,B 0,C 180,E1 -21726.35,E2 -21726.35} C_VEL
LIN {X 0,Y 218.931,Z 696.701,A -85,B 0,C 180,E1 -21727.583,E2 -21727.583} C_VEL
LIN {X 0,Y 221.45,Z 686.448,A -85,B 0,C 180,E1 -21728.667,E2 -21728.667} C_VEL
LIN {X 0,Y 223.828,Z 674.8,A -85,B 0,C 180,E1 -21729.627,E2 -21729.627} C_VEL
LIN {X 0,Y 225.619,Z 663.364,A -85,B 0,C 180,E1 -21730.34,E2 -21730.34} C_VEL
LIN {X 0,Y 226.841,Z 652.577,A -85,B 0,C 180,E1 -21730.822,E2 -21730.822} C_VEL
LIN {X 0,Y 228.511,Z 626.575,A -85,B 0,C 180,E1 -21731.604,E2 -21731.604} C_VEL
LIN {X 0,Y 230.662,Z 586.627,A -85,B 0,C 180,E1 -21732.768,E2 -21732.768} C_VEL
LIN {X 0,Y 229.96,Z 583.237,A -85,B 0,C 180,E1 -21733.07,E2 -21733.07} C_VEL
LIN {X 0,Y 223.645,Z 567.792,A -85,B 0,C 180,E1 -21735.275,E2 -21735.275} C_VEL
LIN {X 0,Y 217.031,Z 554.047,A -85,B 0,C 180,E1 -21737.71,E2 -21737.71} C_VEL
LIN {X 0,Y 209.999,Z 541.266,A -85,B 0,C 180,E1 -21740.514,E2 -21740.514} C_VEL
LIN {X 0,Y 206.178,Z 535.124,A -85,B 0,C 180,E1 -21742.151,E2 -21742.151} C_VEL
LIN {X 0,Y 203.406,Z 530.719,A -85,B 0,C 180,E1 -21743.414,E2 -21743.414} C_VEL
LIN {X 0,Y 200.27,Z 526.105,A -85,B 0,C 180,E1 -21744.911,E2 -21744.911} C_VEL
LIN {X 0,Y 197.67,Z 523.198,A -85,B 0,C 180,E1 -21746.175,E2 -21746.175} C_VEL
LIN {X 0,Y 196.542,Z 521.121,A -85,B 0,C 180,E1 -21746.8,E2 -21746.8} C_VEL
LIN {X 0,Y 194.128,Z 519.133,A -85,B 0,C 180,E1 -21748.032,E2 -21748.032} C_VEL
LIN {X 0,Y 192.744,Z 516.385,A -85,B 0,C 180,E1 -21748.999,E2 -21748.999} C_VEL
LIN {X 0,Y 192.616,Z 515.665,A -85,B 0,C 180,E1 -21749.791,E2 -21749.791} C_VEL
LIN {X 0,Y 192.59,Z 515.594,A -85,B 0,C 180,E1 -21754.029,E2 -21754.029} C_VEL
LIN {X 0,Y 192.683,Z 515.604,A -85,B 0,C 180,E1 -21756.345,E2 -21756.345} C_VEL
LIN {X 0,Y 192.728,Z 515.582,A -85,B 0,C 180,E1 -21761.458,E2 -21761.458} C_VEL
LIN {X 0,Y 192.759,Z 515.564,A -85,B 0,C 180,E1 -21765.212,E2 -21765.212} C_VEL
LIN {X 0,Y 192.978,Z 515.563,A -85,B 0,C 180,E1 -21769.507,E2 -21769.507} C_VEL
LIN {X 0,Y 193.058,Z 515.542,A -85,B 0,C 180,E1 -21771.626,E2 -21771.626} C_VEL
LIN {X 0,Y 193.259,Z 515.534,A -85,B 0,C 180,E1 -21777.915,E2 -21777.915} C_VEL
LIN {X 0,Y 193.439,Z 515.483,A -85,B 0,C 180,E1 -21779.999,E2 -21779.999} C_VEL
LIN {X 0,Y 192.967,Z 515.542,A -85,B 0,C 180,E1 -21784.176,E2 -21784.176} C_VEL
LIN {X 0,Y 193.032,Z 515.529,A -85,B 0,C 180,E1 -21788.373,E2 -21788.373} C_VEL
LIN {X 0,Y 192.796,Z 515.579,A -85,B 0,C 180,E1 -21792.633,E2 -21792.633} C_VEL
LIN {X 0,Y 192.751,Z 515.562,A -85,B 0,C 180,E1 -21796.958,E2 -21796.958} C_VEL
LIN {X 0,Y 192.632,Z 515.611,A -85,B 0,C 180,E1 -21801.397,E2 -21801.397} C_VEL
LIN {X 0,Y 192.659,Z 515.577,A -85,B 0,C 180,E1 -21804.224,E2 -21804.224} C_VEL
LIN {X 0,Y 192.645,Z 515.593,A -85,B 0,C 180,E1 -21808.891,E2 -21808.891} C_VEL
LIN {X 0,Y 192.654,Z 515.885,A -85,B 0,C 180,E1 -21811.091,E2 -21811.091} C_VEL
LIN {X 0,Y 192.977,Z 517.048,A -85,B 0,C 180,E1 -21811.644,E2 -21811.644} C_VEL
LIN {X 0,Y 194.564,Z 519.671,A -85,B 0,C 180,E1 -21812.601,E2 -21812.601} C_VEL
LIN {X 0,Y 196.739,Z 521.387,A -85,B 0,C 180,E1 -21813.697,E2 -21813.697} C_VEL
LIN {X 0,Y 198.842,Z 524.738,A -85,B 0,C 180,E1 -21814.811,E2 -21814.811} C_VEL
LIN {X 0,Y 200.87,Z 526.845,A -85,B 0,C 180,E1 -21815.767,E2 -21815.767} C_VEL
LIN {X 0,Y 203.425,Z 530.373,A -85,B 0,C 180,E1 -21816.966,E2 -21816.966} C_VEL
LIN {X 0,Y 204.836,Z 532.196,A -85,B 0,C 180,E1 -21817.594,E2 -21817.594} C_VEL
LIN {X 0,Y 208.458,Z 537.22,A -85,B 0,C 180,E1 -21819.148,E2 -21819.148} C_VEL
LIN {X 0,Y 213.529,Z 544.449,A -85,B 0,C 180,E1 -21821.167,E2 -21821.167} C_VEL
LIN {X 0,Y 220.054,Z 554.793,A -85,B 0,C 180,E1 -21823.57,E2 -21823.57} C_VEL
LIN {X 0,Y 226.243,Z 565.602,A -85,B 0,C 180,E1 -21825.678,E2 -21825.678} C_VEL
LIN {X 0,Y 235.086,Z 581.768,A -85,B 0,C 180,E1 -21828.412,E2 -21828.412} C_VEL
LIN {X 0,Y 243.356,Z 593.743,A -85,B 0,C 180,E1 -21830.58,E2 -21830.58} C_VEL
LIN {X 0,Y 254.83,Z 607.434,A -85,B 0,C 180,E1 -21833.159,E2 -21833.159} C_VEL
LIN {X 0,Y 272.96,Z 625.122,A -85,B 0,C 180,E1 -21836.529,E2 -21836.529} C_VEL
LIN {X 0,Y 285.856,Z 635.868,A -85,B 0,C 180,E1 -21838.554,E2 -21838.554} C_VEL
LIN {X 0,Y 294.24,Z 642.556,A -85,B 0,C 180,E1 -21839.904,E2 -21839.904} C_VEL
LIN {X 0,Y 302.059,Z 648.597,A -85,B 0,C 180,E1 -21841.352,E2 -21841.352} C_VEL
LIN {X 0,Y 310.022,Z 654.547,A -85,B 0,C 180,E1 -21843.004,E2 -21843.004} C_VEL
LIN {X 0,Y 317.922,Z 660.625,A -85,B 0,C 180,E1 -21844.832,E2 -21844.832} C_VEL
LIN {X 0,Y 324.755,Z 665.526,A -85,B 0,C 180,E1 -21846.55,E2 -21846.55} C_VEL
LIN {X 0,Y 331.943,Z 670.721,A -85,B 0,C 180,E1 -21848.523,E2 -21848.523} C_VEL
LIN {X 0,Y 338.275,Z 675.058,A -85,B 0,C 180,E1 -21850.445,E2 -21850.445} C_VEL
LIN {X 0,Y 343.184,Z 678.721,A -85,B 0,C 180,E1 -21852.111,E2 -21852.111} C_VEL
LIN {X 0,Y 347.08,Z 681.322,A -85,B 0,C 180,E1 -21853.532,E2 -21853.532} C_VEL
LIN {X 0,Y 350.623,Z 683.281,A -85,B 0,C 180,E1 -21854.896,E2 -21854.896} C_VEL
LIN {X 0,Y 354.235,Z 685.648,A -85,B 0,C 180,E1 -21856.444,E2 -21856.444} C_VEL
LIN {X 0,Y 358.432,Z 688.804,A -85,B 0,C 180,E1 -21858.628,E2 -21858.628} C_VEL
LIN {X 0,Y 360.618,Z 690.196,A -85,B 0,C 180,E1 -21859.898,E2 -21859.898} C_VEL
LIN {X 0,Y 364.01,Z 691.956,A -85,B 0,C 180,E1 -21862.233,E2 -21862.233} C_VEL
LIN {X 0,Y 366.506,Z 693.154,A -85,B 0,C 180,E1 -21864.498,E2 -21864.498} C_VEL
LIN {X 0,Y 368.185,Z 693.703,A -85,B 0,C 180,E1 -21866.717,E2 -21866.717} C_VEL
LIN {X 0,Y 368.945,Z 694.133,A -85,B 0,C 180,E1 -21868.909,E2 -21868.909} C_VEL
LIN {X 0,Y 369.086,Z 694.049,A -85,B 0,C 180,E1 -21870,E2 -21870} C_VEL
LIN {X 0,Y 368.65,Z 693.959,A -85,B 0,C 180,E1 -21872.185,E2 -21872.185} C_VEL
LIN {X 0,Y 367.422,Z 693.486,A -85,B 0,C 180,E1 -21874.388,E2 -21874.388} C_VEL
LIN {X 0,Y 365.379,Z 692.617,A -85,B 0,C 180,E1 -21876.627,E2 -21876.627} C_VEL
LIN {X 0,Y 362.663,Z 691.299,A -85,B 0,C 180,E1 -21878.77,E2 -21878.77} C_VEL
LIN {X 0,Y 360.623,Z 690.124,A -85,B 0,C 180,E1 -21880.101,E2 -21880.101} C_VEL
LIN {X 0,Y 358.442,Z 688.791,A -85,B 0,C 180,E1 -21881.38,E2 -21881.38} C_VEL
LIN {X 0,Y 354.226,Z 685.661,A -85,B 0,C 180,E1 -21883.55,E2 -21883.55} C_VEL
LIN {X 0,Y 349.914,Z 682.885,A -85,B 0,C 180,E1 -21885.407,E2 -21885.407} C_VEL
LIN {X 0,Y 345.522,Z 680.268,A -85,B 0,C 180,E1 -21887.064,E2 -21887.064} C_VEL
LIN {X 0,Y 339.521,Z 676.055,A -85,B 0,C 180,E1 -21889.129,E2 -21889.129} C_VEL
LIN {X 0,Y 335.274,Z 672.925,A -85,B 0,C 180,E1 -21890.489,E2 -21890.489} C_VEL
LIN {X 0,Y 329.355,Z 669.022,A -85,B 0,C 180,E1 -21892.194,E2 -21892.194} C_VEL
LIN {X 0,Y 321.641,Z 663.231,A -85,B 0,C 180,E1 -21894.252,E2 -21894.252} C_VEL
LIN {X 0,Y 313.882,Z 657.603,A -85,B 0,C 180,E1 -21896.12,E2 -21896.12} C_VEL
LIN {X 0,Y 306.85,Z 652.291,A -85,B 0,C 180,E1 -21897.664,E2 -21897.664} C_VEL
LIN {X 0,Y 299.011,Z 646.098,A -85,B 0,C 180,E1 -21899.24,E2 -21899.24} C_VEL
LIN {X 0,Y 290.318,Z 639.473,A -85,B 0,C 180,E1 -21900.755,E2 -21900.755} C_VEL
LIN {X 0,Y 276.6,Z 628.236,A -85,B 0,C 180,E1 -21902.875,E2 -21902.875} C_VEL
LIN {X 0,Y 262.126,Z 614.903,A -85,B 0,C 180,E1 -21905.4,E2 -21905.4} C_VEL
LIN {X 0,Y 249.189,Z 601.029,A -85,B 0,C 180,E1 -21908.056,E2 -21908.056} C_VEL
LIN {X 0,Y 239.26,Z 588.151,A -85,B 0,C 180,E1 -21910.453,E2 -21910.453} C_VEL
LIN {X 0,Y 231.554,Z 575.709,A -85,B 0,C 180,E1 -21912.624,E2 -21912.624} C_VEL
LIN {X 0,Y 223.27,Z 560.238,A -85,B 0,C 180,E1 -21915.318,E2 -21915.318} C_VEL
LIN {X 0,Y 216.084,Z 548.302,A -85,B 0,C 180,E1 -21917.871,E2 -21917.871} C_VEL
LIN {X 0,Y 209.417,Z 538.503,A -85,B 0,C 180,E1 -21920.46,E2 -21920.46} C_VEL
LIN {X 0,Y 206.007,Z 533.851,A -85,B 0,C 180,E1 -21921.89,E2 -21921.89} C_VEL
LIN {X 0,Y 203.545,Z 530.494,A -85,B 0,C 180,E1 -21922.982,E2 -21922.982} C_VEL
LIN {X 0,Y 200.867,Z 526.871,A -85,B 0,C 180,E1 -21924.232,E2 -21924.232} C_VEL
LIN {X 0,Y 197.553,Z 522.974,A -85,B 0,C 180,E1 -21925.847,E2 -21925.847} C_VEL
LIN {X 0,Y 196.411,Z 521.045,A -85,B 0,C 180,E1 -21926.47,E2 -21926.47} C_VEL
LIN {X 0,Y 194.146,Z 519.156,A -85,B 0,C 180,E1 -21927.629,E2 -21927.629} C_VEL
LIN {X 0,Y 192.732,Z 516.161,A -85,B 0,C 180,E1 -21928.694,E2 -21928.694} C_VEL
LIN {X 0,Y 192.622,Z 515.647,A -85,B 0,C 180,E1 -21929.284,E2 -21929.284} C_VEL
LIN {X 0,Y 192.66,Z 515.6,A -85,B 0,C 180,E1 -21931.692,E2 -21931.692} C_VEL
LIN {X 0,Y 192.701,Z 515.573,A -85,B 0,C 180,E1 -21936.349,E2 -21936.349} C_VEL
LIN {X 0,Y 192.727,Z 515.569,A -85,B 0,C 180,E1 -21941.459,E2 -21941.459} C_VEL
LIN {X 0,Y 192.756,Z 515.586,A -85,B 0,C 180,E1 -21945.214,E2 -21945.214} C_VEL
LIN {X 0,Y 192.941,Z 515.534,A -85,B 0,C 180,E1 -21949.567,E2 -21949.567} C_VEL
LIN {X 0,Y 192.982,Z 515.569,A -85,B 0,C 180,E1 -21953.729,E2 -21953.729} C_VEL
LIN {X 0,Y 193.258,Z 515.489,A -85,B 0,C 180,E1 -21957.917,E2 -21957.917} C_VEL
LIN {X 0,Y 193.439,Z 515.483,A -85,B 0,C 180,E1 -21960.001,E2 -21960.001} C_VEL
LIN {X 0,Y 192.971,Z 515.536,A -85,B 0,C 180,E1 -21964.178,E2 -21964.178} C_VEL
LIN {X 0,Y 193.058,Z 515.542,A -85,B 0,C 180,E1 -21968.374,E2 -21968.374} C_VEL
LIN {X 0,Y 192.806,Z 515.554,A -85,B 0,C 180,E1 -21972.634,E2 -21972.634} C_VEL
LIN {X 0,Y 192.754,Z 515.599,A -85,B 0,C 180,E1 -21976.96,E2 -21976.96} C_VEL
LIN {X 0,Y 192.612,Z 515.582,A -85,B 0,C 180,E1 -21981.401,E2 -21981.401} C_VEL
LIN {X 0,Y 192.645,Z 515.613,A -85,B 0,C 180,E1 -21984.214,E2 -21984.214} C_VEL
LIN {X 0,Y 192.643,Z 515.592,A -85,B 0,C 180,E1 -21988.89,E2 -21988.89} C_VEL
LIN {X 0,Y 192.663,Z 515.931,A -85,B 0,C 180,E1 -21990.711,E2 -21990.711} C_VEL
LIN {X 0,Y 192.988,Z 517.104,A -85,B 0,C 180,E1 -21991.262,E2 -21991.262} C_VEL
LIN {X 0,Y 194.542,Z 519.629,A -85,B 0,C 180,E1 -21992.195,E2 -21992.195} C_VEL
LIN {X 0,Y 196.754,Z 521.412,A -85,B 0,C 180,E1 -21993.313,E2 -21993.313} C_VEL
LIN {X 0,Y 198.648,Z 524.523,A -85,B 0,C 180,E1 -21994.324,E2 -21994.324} C_VEL
LIN {X 0,Y 200.822,Z 526.787,A -85,B 0,C 180,E1 -21995.352,E2 -21995.352} C_VEL
LIN {X 0,Y 204.901,Z 533.043,A -85,B 0,C 180,E1 -21997.273,E2 -21997.273} C_VEL
LIN {X 0,Y 210.503,Z 542.137,A -85,B 0,C 180,E1 -21999.696,E2 -21999.696} C_VEL
LIN {X 0,Y 217.513,Z 555.016,A -85,B 0,C 180,E1 -22002.475,E2 -22002.475} C_VEL
LIN {X 0,Y 223.119,Z 566.726,A -85,B 0,C 180,E1 -22004.541,E2 -22004.541} C_VEL
LIN {X 0,Y 228.923,Z 580.563,A -85,B 0,C 180,E1 -22006.576,E2 -22006.576} C_VEL
LIN {X 0,Y 230.34,Z 584.699,A -85,B 0,C 180,E1 -22007.078,E2 -22007.078} C_VEL
LIN {X 0,Y 230.681,Z 587.988,A -85,B 0,C 180,E1 -22007.292,E2 -22007.292} C_VEL
LIN {X 0,Y 226.97,Z 651.29,A -85,B 0,C 180,E1 -22009.128,E2 -22009.128} C_VEL
LIN {X 0,Y 225.761,Z 662.453,A -85,B 0,C 180,E1 -22009.618,E2 -22009.618} C_VEL
LIN {X 0,Y 224.084,Z 673.441,A -85,B 0,C 180,E1 -22010.282,E2 -22010.282} C_VEL
LIN {X 0,Y 222.112,Z 683.228,A -85,B 0,C 180,E1 -22011.034,E2 -22011.034} C_VEL
LIN {X 0,Y 219.869,Z 693.197,A -85,B 0,C 180,E1 -22012.026,E2 -22012.026} C_VEL
LIN {X 0,Y 217.254,Z 703.113,A -85,B 0,C 180,E1 -22013.241,E2 -22013.241} C_VEL
LIN {X 0,Y 214.209,Z 713.021,A -85,B 0,C 180,E1 -22014.717,E2 -22014.717} C_VEL
LIN {X 0,Y 211.159,Z 722.43,A -85,B 0,C 180,E1 -22016.453,E2 -22016.453} C_VEL
LIN {X 0,Y 207.984,Z 731.271,A -85,B 0,C 180,E1 -22018.416,E2 -22018.416} C_VEL
LIN {X 0,Y 205.998,Z 736.381,A -85,B 0,C 180,E1 -22019.694,E2 -22019.694} C_VEL
LIN {X 0,Y 203.807,Z 740.426,A -85,B 0,C 180,E1 -22020.731,E2 -22020.731} C_VEL
LIN {X 0,Y 198.579,Z 746.549,A -85,B 0,C 180,E1 -22022.383,E2 -22022.383} C_VEL
LIN {X 0,Y 193.425,Z 752.264,A -85,B 0,C 180,E1 -22024.239,E2 -22024.239} C_VEL
LIN {X 0,Y 191.385,Z 755.41,A -85,B 0,C 180,E1 -22025.58,E2 -22025.58} C_VEL
LIN {X 0,Y 188.228,Z 762.691,A -85,B 0,C 180,E1 -22029.416,E2 -22029.416} C_VEL
LIN {X 0,Y 185.788,Z 768.465,A -85,B 0,C 180,E1 -22033.519,E2 -22033.519} C_VEL
LIN {X 0,Y 184.368,Z 772.014,A -85,B 0,C 180,E1 -22036.779,E2 -22036.779} C_VEL
LIN {X 0,Y 183.806,Z 773.962,A -85,B 0,C 180,E1 -22038.979,E2 -22038.979} C_VEL
LIN {X 0,Y 183.137,Z 776.658,A -85,B 0,C 180,E1 -22043.389,E2 -22043.389} C_VEL
LIN {X 0,Y 183.055,Z 777.804,A -85,B 0,C 180,E1 -22046.586,E2 -22046.586} C_VEL
LIN {X 0,Y 183.172,Z 778.217,A -85,B 0,C 180,E1 -22050,E2 -22050} C_VEL
LIN {X 0,Y 183.076,Z 777.483,A -85,B 0,C 180,E1 -22054.403,E2 -22054.403} C_VEL
LIN {X 0,Y 183.137,Z 776.658,A -85,B 0,C 180,E1 -22056.611,E2 -22056.611} C_VEL
LIN {X 0,Y 183.806,Z 773.962,A -85,B 0,C 180,E1 -22061.021,E2 -22061.021} C_VEL
LIN {X 0,Y 185.244,Z 769.733,A -85,B 0,C 180,E1 -22065.401,E2 -22065.401} C_VEL
LIN {X 0,Y 186.942,Z 765.596,A -85,B 0,C 180,E1 -22068.636,E2 -22068.636} C_VEL
LIN {X 0,Y 189.095,Z 760.491,A -85,B 0,C 180,E1 -22071.818,E2 -22071.818} C_VEL
LIN {X 0,Y 191.859,Z 754.312,A -85,B 0,C 180,E1 -22074.913,E2 -22074.913} C_VEL
LIN {X 0,Y 194.592,Z 748.238,A -85,B 0,C 180,E1 -22077.418,E2 -22077.418} C_VEL
LIN {X 0,Y 197.639,Z 741.164,A -85,B 0,C 180,E1 -22079.856,E2 -22079.856} C_VEL
LIN {X 0,Y 200.485,Z 734.708,A -85,B 0,C 180,E1 -22081.723,E2 -22081.723} C_VEL
LIN {X 0,Y 204.482,Z 724.498,A -85,B 0,C 180,E1 -22084.158,E2 -22084.158} C_VEL
LIN {X 0,Y 207.727,Z 715.115,A -85,B 0,C 180,E1 -22086.003,E2 -22086.003} C_VEL
LIN {X 0,Y 210.699,Z 705.842,A -85,B 0,C 180,E1 -22087.497,E2 -22087.497} C_VEL
LIN {X 0,Y 213.354,Z 696.503,A -85,B 0,C 180,E1 -22088.745,E2 -22088.745} C_VEL
LIN {X 0,Y 215.953,Z 686.25,A -85,B 0,C 180,E1 -22089.844,E2 -22089.844} C_VEL
LIN {X 0,Y 218.397,Z 674.601,A -85,B 0,C 180,E1 -22090.817,E2 -22090.817} C_VEL
LIN {X 0,Y 220.262,Z 663.166,A -85,B 0,C 180,E1 -22091.534,E2 -22091.534} C_VEL
LIN {X 0,Y 221.494,Z 652.73,A -85,B 0,C 180,E1 -22092.008,E2 -22092.008} C_VEL
LIN {X 0,Y 222.952,Z 631.299,A -85,B 0,C 180,E1 -22092.674,E2 -22092.674} C_VEL
LIN {X 0,Y 225.392,Z 587.492,A -85,B 0,C 180,E1 -22093.974,E2 -22093.974} C_VEL
LIN {X 0,Y 219.946,Z 573.53,A -85,B 0,C 180,E1 -22095.986,E2 -22095.986} C_VEL
LIN {X 0,Y 213.657,Z 559.959,A -85,B 0,C 180,E1 -22098.414,E2 -22098.414} C_VEL
LIN {X 0,Y 207.095,Z 547.629,A -85,B 0,C 180,E1 -22101.149,E2 -22101.149} C_VEL
LIN {X 0,Y 202.673,Z 540.174,A -85,B 0,C 180,E1 -22103.144,E2 -22103.144} C_VEL
LIN {X 0,Y 199.785,Z 535.588,A -85,B 0,C 180,E1 -22104.531,E2 -22104.531} C_VEL
LIN {X 0,Y 197.387,Z 532.045,A -85,B 0,C 180,E1 -22105.735,E2 -22105.735} C_VEL
LIN {X 0,Y 194.574,Z 528.553,A -85,B 0,C 180,E1 -22107.193,E2 -22107.193} C_VEL
LIN {X 0,Y 193.674,Z 527.222,A -85,B 0,C 180,E1 -22107.695,E2 -22107.695} C_VEL
LIN {X 0,Y 191.142,Z 524.568,A -85,B 0,C 180,E1 -22109.095,E2 -22109.095} C_VEL
LIN {X 0,Y 189.721,Z 522.129,A -85,B 0,C 180,E1 -22109.993,E2 -22109.993} C_VEL
LIN {X 0,Y 187.137,Z 520.056,A -85,B 0,C 180,E1 -22111.543,E2 -22111.543} C_VEL
LIN {X 0,Y 185.65,Z 517.1,A -85,B 0,C 180,E1 -22112.828,E2 -22112.828} C_VEL
LIN {X 0,Y 185.569,Z 516.528,A -85,B 0,C 180,E1 -22113.576,E2 -22113.576} C_VEL
LIN {X 0,Y 185.575,Z 516.465,A -85,B 0,C 180,E1 -22117.745,E2 -22117.745} C_VEL
LIN {X 0,Y 185.686,Z 516.474,A -85,B 0,C 180,E1 -22122.374,E2 -22122.374} C_VEL
LIN {X 0,Y 185.73,Z 516.433,A -85,B 0,C 180,E1 -22126.876,E2 -22126.876} C_VEL
LIN {X 0,Y 186.005,Z 516.425,A -85,B 0,C 180,E1 -22131.306,E2 -22131.306} C_VEL
LIN {X 0,Y 186.203,Z 516.411,A -85,B 0,C 180,E1 -22137.836,E2 -22137.836} C_VEL
LIN {X 0,Y 186.402,Z 516.358,A -85,B 0,C 180,E1 -22139.999,E2 -22139.999} C_VEL
LIN {X 0,Y 185.913,Z 516.421,A -85,B 0,C 180,E1 -22144.335,E2 -22144.335} C_VEL
LIN {X 0,Y 185.978,Z 516.404,A -85,B 0,C 180,E1 -22148.693,E2 -22148.693} C_VEL
LIN {X 0,Y 185.723,Z 516.468,A -85,B 0,C 180,E1 -22153.122,E2 -22153.122} C_VEL
LIN {X 0,Y 185.685,Z 516.441,A -85,B 0,C 180,E1 -22157.624,E2 -22157.624} C_VEL
LIN {X 0,Y 185.592,Z 516.471,A -85,B 0,C 180,E1 -22162.251,E2 -22162.251} C_VEL
LIN {X 0,Y 185.57,Z 516.642,A -85,B 0,C 180,E1 -22167.03,E2 -22167.03} C_VEL
LIN {X 0,Y 185.808,Z 517.598,A -85,B 0,C 180,E1 -22167.831,E2 -22167.831} C_VEL
LIN {X 0,Y 187.427,Z 520.422,A -85,B 0,C 180,E1 -22169.039,E2 -22169.039} C_VEL
LIN {X 0,Y 190.008,Z 522.409,A -85,B 0,C 180,E1 -22170.568,E2 -22170.568} C_VEL
LIN {X 0,Y 191.892,Z 525.606,A -85,B 0,C 180,E1 -22171.74,E2 -22171.74} C_VEL
LIN {X 0,Y 194.262,Z 527.964,A -85,B 0,C 180,E1 -22173.019,E2 -22173.019} C_VEL
LIN {X 0,Y 196.922,Z 531.615,A -85,B 0,C 180,E1 -22174.432,E2 -22174.432} C_VEL
LIN {X 0,Y 198.159,Z 533.034,A -85,B 0,C 180,E1 -22175.043,E2 -22175.043} C_VEL
LIN {X 0,Y 201.088,Z 536.856,A -85,B 0,C 180,E1 -22176.451,E2 -22176.451} C_VEL
LIN {X 0,Y 207.629,Z 546.228,A -85,B 0,C 180,E1 -22179.35,E2 -22179.35} C_VEL
LIN {X 0,Y 214.12,Z 556.277,A -85,B 0,C 180,E1 -22181.935,E2 -22181.935} C_VEL
LIN {X 0,Y 221.362,Z 568.872,A -85,B 0,C 180,E1 -22184.571,E2 -22184.571} C_VEL
LIN {X 0,Y 230.397,Z 585.785,A -85,B 0,C 180,E1 -22187.529,E2 -22187.529} C_VEL
LIN {X 0,Y 238.94,Z 598.519,A -85,B 0,C 180,E1 -22189.883,E2 -22189.883} C_VEL
LIN {X 0,Y 250.506,Z 612.496,A -85,B 0,C 180,E1 -22192.589,E2 -22192.589} C_VEL
LIN {X 0,Y 267.863,Z 629.71,A -85,B 0,C 180,E1 -22195.946,E2 -22195.946} C_VEL
LIN {X 0,Y 281.844,Z 641.539,A -85,B 0,C 180,E1 -22198.252,E2 -22198.252} C_VEL
LIN {X 0,Y 291.736,Z 649.424,A -85,B 0,C 180,E1 -22199.889,E2 -22199.889} C_VEL
LIN {X 0,Y 299.865,Z 655.716,A -85,B 0,C 180,E1 -22201.42,E2 -22201.42} C_VEL
LIN {X 0,Y 308.442,Z 662.127,A -85,B 0,C 180,E1 -22203.227,E2 -22203.227} C_VEL
LIN {X 0,Y 316.086,Z 667.871,A -85,B 0,C 180,E1 -22205.011,E2 -22205.011} C_VEL
LIN {X 0,Y 321.926,Z 672.076,A -85,B 0,C 180,E1 -22206.476,E2 -22206.476} C_VEL
LIN {X 0,Y 328.38,Z 676.789,A -85,B 0,C 180,E1 -22208.263,E2 -22208.263} C_VEL
LIN {X 0,Y 335.644,Z 681.716,A -85,B 0,C 180,E1 -22210.43,E2 -22210.43} C_VEL
LIN {X 0,Y 340.116,Z 685.025,A -85,B 0,C 180,E1 -22211.944,E2 -22211.944} C_VEL
LIN {X 0,Y 344.456,Z 687.912,A -85,B 0,C 180,E1 -22213.523,E2 -22213.523} C_VEL
LIN {X 0,Y 348.856,Z 690.425,A -85,B 0,C 180,E1 -22215.237,E2 -22215.237} C_VEL
LIN {X 0,Y 350.812,Z 691.681,A -85,B 0,C 180,E1 -22216.09,E2 -22216.09} C_VEL
LIN {X 0,Y 353.346,Z 693.708,A -85,B 0,C 180,E1 -22217.362,E2 -22217.362} C_VEL
LIN {X 0,Y 357.31,Z 696.383,A -85,B 0,C 180,E1 -22219.561,E2 -22219.561} C_VEL
LIN {X 0,Y 359.56,Z 697.629,A -85,B 0,C 180,E1 -22221.004,E2 -22221.004} C_VEL
LIN {X 0,Y 362.565,Z 699.145,A -85,B 0,C 180,E1 -22223.321,E2 -22223.321} C_VEL
LIN {X 0,Y 364.708,Z 700.021,A -85,B 0,C 180,E1 -22225.579,E2 -22225.579} C_VEL
LIN {X 0,Y 365.966,Z 700.504,A -85,B 0,C 180,E1 -22227.799,E2 -22227.799} C_VEL
LIN {X 0,Y 366.407,Z 700.605,A -85,B 0,C 180,E1 -22230,E2 -22230} C_VEL
LIN {X 0,Y 365.944,Z 700.521,A -85,B 0,C 180,E1 -22232.201,E2 -22232.201} C_VEL
LIN {X 0,Y 365.448,Z 700.248,A -85,B 0,C 180,E1 -22233.307,E2 -22233.307} C_VEL
LIN {X 0,Y 363.712,Z 699.653,A -85,B 0,C 180,E1 -22235.544,E2 -22235.544} C_VEL
LIN {X 0,Y 361.172,Z 698.501,A -85,B 0,C 180,E1 -22237.829,E2 -22237.829} C_VEL
LIN {X 0,Y 359.579,Z 697.623,A -85,B 0,C 180,E1 -22238.995,E2 -22238.995} C_VEL
LIN {X 0,Y 357.307,Z 696.333,A -85,B 0,C 180,E1 -22240.437,E2 -22240.437} C_VEL
LIN {X 0,Y 353.378,Z 693.696,A -85,B 0,C 180,E1 -22242.636,E2 -22242.636} C_VEL
LIN {X 0,Y 350.797,Z 691.674,A -85,B 0,C 180,E1 -22243.911,E2 -22243.911} C_VEL
LIN {X 0,Y 347.72,Z 689.706,A -85,B 0,C 180,E1 -22245.233,E2 -22245.233} C_VEL
LIN {X 0,Y 342.389,Z 686.573,A -85,B 0,C 180,E1 -22247.225,E2 -22247.225} C_VEL
LIN {X 0,Y 337.706,Z 683.322,A -85,B 0,C 180,E1 -22248.876,E2 -22248.876} C_VEL
LIN {X 0,Y 334.007,Z 680.416,A -85,B 0,C 180,E1 -22250.09,E2 -22250.09} C_VEL
LIN {X 0,Y 326.518,Z 675.551,A -85,B 0,C 180,E1 -22252.253,E2 -22252.253} C_VEL
LIN {X 0,Y 319.666,Z 670.28,A -85,B 0,C 180,E1 -22254.113,E2 -22254.113} C_VEL
LIN {X 0,Y 311.93,Z 664.822,A -85,B 0,C 180,E1 -22255.972,E2 -22255.972} C_VEL
LIN {X 0,Y 304.274,Z 659.029,A -85,B 0,C 180,E1 -22257.678,E2 -22257.678} C_VEL
LIN {X 0,Y 295.53,Z 652.236,A -85,B 0,C 180,E1 -22259.429,E2 -22259.429} C_VEL
LIN {X 0,Y 286.642,Z 645.466,A -85,B 0,C 180,E1 -22260.97,E2 -22260.97} C_VEL
LIN {X 0,Y 272.622,Z 633.843,A -85,B 0,C 180,E1 -22263.248,E2 -22263.248} C_VEL
LIN {X 0,Y 258.458,Z 620.733,A -85,B 0,C 180,E1 -22265.788,E2 -22265.788} C_VEL
LIN {X 0,Y 245.663,Z 606.934,A -85,B 0,C 180,E1 -22268.49,E2 -22268.49} C_VEL
LIN {X 0,Y 235.337,Z 593.516,A -85,B 0,C 180,E1 -22271.064,E2 -22271.064} C_VEL
LIN {X 0,Y 227.834,Z 581.292,A -85,B 0,C 180,E1 -22273.259,E2 -22273.259} C_VEL
LIN {X 0,Y 218.733,Z 564.131,A -85,B 0,C 180,E1 -22276.359,E2 -22276.359} C_VEL
LIN {X 0,Y 211.374,Z 551.872,A -85,B 0,C 180,E1 -22279.13,E2 -22279.13} C_VEL
LIN {X 0,Y 204.095,Z 541.029,A -85,B 0,C 180,E1 -22282.177,E2 -22282.177} C_VEL
LIN {X 0,Y 199.98,Z 535.65,A -85,B 0,C 180,E1 -22284.057,E2 -22284.057} C_VEL
LIN {X 0,Y 197.262,Z 531.932,A -85,B 0,C 180,E1 -22285.403,E2 -22285.403} C_VEL
LIN {X 0,Y 194.526,Z 528.433,A -85,B 0,C 180,E1 -22286.83,E2 -22286.83} C_VEL
LIN {X 0,Y 193.777,Z 527.284,A -85,B 0,C 180,E1 -22287.25,E2 -22287.25} C_VEL
LIN {X 0,Y 191.311,Z 524.794,A -85,B 0,C 180,E1 -22288.602,E2 -22288.602} C_VEL
LIN {X 0,Y 189.812,Z 522.163,A -85,B 0,C 180,E1 -22289.551,E2 -22289.551} C_VEL
LIN {X 0,Y 187.345,Z 520.328,A -85,B 0,C 180,E1 -22291.013,E2 -22291.013} C_VEL
LIN {X 0,Y 185.704,Z 517.163,A -85,B 0,C 180,E1 -22292.381,E2 -22292.381} C_VEL
LIN {X 0,Y 185.551,Z 516.506,A -85,B 0,C 180,E1 -22293.576,E2 -22293.576} C_VEL
LIN {X 0,Y 185.592,Z 516.471,A -85,B 0,C 180,E1 -22297.749,E2 -22297.749} C_VEL
LIN {X 0,Y 185.685,Z 516.441,A -85,B 0,C 180,E1 -22302.376,E2 -22302.376} C_VEL
LIN {X 0,Y 185.723,Z 516.468,A -85,B 0,C 180,E1 -22306.878,E2 -22306.878} C_VEL
LIN {X 0,Y 185.979,Z 516.404,A -85,B 0,C 180,E1 -22311.307,E2 -22311.307} C_VEL
LIN {X 0,Y 186.202,Z 516.368,A -85,B 0,C 180,E1 -22317.838,E2 -22317.838} C_VEL
LIN {X 0,Y 186.402,Z 516.358,A -85,B 0,C 180,E1 -22320.001,E2 -22320.001} C_VEL
LIN {X 0,Y 185.918,Z 516.412,A -85,B 0,C 180,E1 -22324.337,E2 -22324.337} C_VEL
LIN {X 0,Y 186.005,Z 516.425,A -85,B 0,C 180,E1 -22328.694,E2 -22328.694} C_VEL
LIN {X 0,Y 185.73,Z 516.433,A -85,B 0,C 180,E1 -22333.124,E2 -22333.124} C_VEL
LIN {X 0,Y 185.686,Z 516.474,A -85,B 0,C 180,E1 -22337.626,E2 -22337.626} C_VEL
LIN {X 0,Y 185.575,Z 516.465,A -85,B 0,C 180,E1 -22342.255,E2 -22342.255} C_VEL
LIN {X 0,Y 185.583,Z 516.702,A -85,B 0,C 180,E1 -22346.801,E2 -22346.801} C_VEL
LIN {X 0,Y 185.868,Z 517.816,A -85,B 0,C 180,E1 -22347.518,E2 -22347.518} C_VEL
LIN {X 0,Y 187.431,Z 520.405,A -85,B 0,C 180,E1 -22348.648,E2 -22348.648} C_VEL
LIN {X 0,Y 190.013,Z 522.508,A -85,B 0,C 180,E1 -22350.186,E2 -22350.186} C_VEL
LIN {X 0,Y 192.08,Z 525.775,A -85,B 0,C 180,E1 -22351.45,E2 -22351.45} C_VEL
LIN {X 0,Y 194.099,Z 527.684,A -85,B 0,C 180,E1 -22352.533,E2 -22352.533} C_VEL
LIN {X 0,Y 196.492,Z 531.128,A -85,B 0,C 180,E1 -22353.824,E2 -22353.824} C_VEL
LIN {X 0,Y 198.16,Z 533.039,A -85,B 0,C 180,E1 -22354.651,E2 -22354.651} C_VEL
LIN {X 0,Y 201.934,Z 538.977,A -85,B 0,C 180,E1 -22356.508,E2 -22356.508} C_VEL
LIN {X 0,Y 207.094,Z 547.637,A -85,B 0,C 180,E1 -22358.852,E2 -22358.852} C_VEL
LIN {X 0,Y 213.586,Z 559.796,A -85,B 0,C 180,E1 -22361.557,E2 -22361.557} C_VEL
LIN {X 0,Y 219.31,Z 572.159,A -85,B 0,C 180,E1 -22363.78,E2 -22363.78} C_VEL
LIN {X 0,Y 224.436,Z 584.731,A -85,B 0,C 180,E1 -22365.671,E2 -22365.671} C_VEL
LIN {X 0,Y 225.421,Z 587.99,A -85,B 0,C 180,E1 -22366.055,E2 -22366.055} C_VEL
LIN {X 0,Y 221.725,Z 650.24,A -85,B 0,C 180,E1 -22367.894,E2 -22367.894} C_VEL
LIN {X 0,Y 220.409,Z 662.255,A -85,B 0,C 180,E1 -22368.424,E2 -22368.424} C_VEL
LIN {X 0,Y 218.675,Z 673.243,A -85,B 0,C 180,E1 -22369.094,E2 -22369.094} C_VEL
LIN {X 0,Y 216.649,Z 683.03,A -85,B 0,C 180,E1 -22369.855,E2 -22369.855} C_VEL
LIN {X 0,Y 214.316,Z 692.998,A -85,B 0,C 180,E1 -22370.858,E2 -22370.858} C_VEL
LIN {X 0,Y 211.598,Z 702.915,A -85,B 0,C 180,E1 -22372.088,E2 -22372.088} C_VEL
LIN {X 0,Y 208.492,Z 712.633,A -85,B 0,C 180,E1 -22373.551,E2 -22373.551} C_VEL
LIN {X 0,Y 205.225,Z 722.23,A -85,B 0,C 180,E1 -22375.348,E2 -22375.348} C_VEL
LIN {X 0,Y 201.94,Z 731.072,A -85,B 0,C 180,E1 -22377.356,E2 -22377.356} C_VEL
LIN {X 0,Y 199.047,Z 738.043,A -85,B 0,C 180,E1 -22379.206,E2 -22379.206} C_VEL
LIN {X 0,Y 195.786,Z 745.563,A -85,B 0,C 180,E1 -22381.601,E2 -22381.601} C_VEL
LIN {X 0,Y 192.929,Z 752.037,A -85,B 0,C 180,E1 -22384.079,E2 -22384.079} C_VEL
LIN {X 0,Y 191.385,Z 755.41,A -85,B 0,C 180,E1 -22385.58,E2 -22385.58} C_VEL
LIN {X 0,Y 189.441,Z 758.478,A -85,B 0,C 180,E1 -22386.983,E2 -22386.983} C_VEL
LIN {X 0,Y 184.723,Z 762.973,A -85,B 0,C 180,E1 -22389.273,E2 -22389.273} C_VEL
LIN {X 0,Y 180.208,Z 766.922,A -85,B 0,C 180,E1 -22391.771,E2 -22391.771} C_VEL
LIN {X 0,Y 178.633,Z 768.942,A -85,B 0,C 180,E1 -22393.466,E2 -22393.466} C_VEL
LIN {X 0,Y 177.409,Z 771.815,A -85,B 0,C 180,E1 -22396.25,E2 -22396.25} C_VEL
LIN {X 0,Y 176.795,Z 773.762,A -85,B 0,C 180,E1 -22398.536,E2 -22398.536} C_VEL
LIN {X 0,Y 176.079,Z 776.46,A -85,B 0,C 180,E1 -22403.123,E2 -22403.123} C_VEL
LIN {X 0,Y 175.972,Z 777.763,A -85,B 0,C 180,E1 -22407.711,E2 -22407.711} C_VEL
LIN {X 0,Y 176.079,Z 778.019,A -85,B 0,C 180,E1 -22410,E2 -22410} C_VEL
LIN {X 0,Y 175.973,Z 777.284,A -85,B 0,C 180,E1 -22414.581,E2 -22414.581} C_VEL
LIN {X 0,Y 176.079,Z 776.46,A -85,B 0,C 180,E1 -22416.877,E2 -22416.877} C_VEL
LIN {X 0,Y 176.795,Z 773.762,A -85,B 0,C 180,E1 -22421.464,E2 -22421.464} C_VEL
LIN {X 0,Y 178.38,Z 769.534,A -85,B 0,C 180,E1 -22426.009,E2 -22426.009} C_VEL
LIN {X 0,Y 180.182,Z 765.396,A -85,B 0,C 180,E1 -22429.362,E2 -22429.362} C_VEL
LIN {X 0,Y 182.488,Z 760.292,A -85,B 0,C 180,E1 -22432.651,E2 -22432.651} C_VEL
LIN {X 0,Y 185.407,Z 754.113,A -85,B 0,C 180,E1 -22435.843,E2 -22435.843} C_VEL
LIN {X 0,Y 188.283,Z 748.039,A -85,B 0,C 180,E1 -22438.418,E2 -22438.418} C_VEL
LIN {X 0,Y 191.5,Z 740.965,A -85,B 0,C 180,E1 -22440.916,E2 -22440.916} C_VEL
LIN {X 0,Y 194.462,Z 734.51,A -85,B 0,C 180,E1 -22442.827,E2 -22442.827} C_VEL
LIN {X 0,Y 198.474,Z 724.704,A -85,B 0,C 180,E1 -22445.224,E2 -22445.224} C_VEL
LIN {X 0,Y 201.574,Z 716.156,A -85,B 0,C 180,E1 -22446.972,E2 -22446.972} C_VEL
LIN {X 0,Y 204.643,Z 707.108,A -85,B 0,C 180,E1 -22448.495,E2 -22448.495} C_VEL
LIN {X 0,Y 207.862,Z 696.305,A -85,B 0,C 180,E1 -22449.97,E2 -22449.97} C_VEL
LIN {X 0,Y 210.548,Z 686.052,A -85,B 0,C 180,E1 -22451.083,E2 -22451.083} C_VEL
LIN {X 0,Y 213.075,Z 674.403,A -85,B 0,C 180,E1 -22452.064,E2 -22452.064} C_VEL
LIN {X 0,Y 214.991,Z 662.968,A -85,B 0,C 180,E1 -22452.79,E2 -22452.79} C_VEL
LIN {X 0,Y 216.342,Z 651.645,A -85,B 0,C 180,E1 -22453.302,E2 -22453.302} C_VEL
LIN {X 0,Y 217.985,Z 628.061,A -85,B 0,C 180,E1 -22454.026,E2 -22454.026} C_VEL
LIN {X 0,Y 220.272,Z 589.664,A -85,B 0,C 180,E1 -22455.166,E2 -22455.166} C_VEL
LIN {X 0,Y 214.765,Z 575.647,A -85,B 0,C 180,E1 -22457.324,E2 -22457.324} C_VEL
LIN {X 0,Y 208.68,Z 562.518,A -85,B 0,C 180,E1 -22459.834,E2 -22459.834} C_VEL
LIN {X 0,Y 202.61,Z 551.032,A -85,B 0,C 180,E1 -22462.546,E2 -22462.546} C_VEL
LIN {X 0,Y 197.272,Z 541.976,A -85,B 0,C 180,E1 -22465.162,E2 -22465.162} C_VEL
LIN {X 0,Y 194.462,Z 537.844,A -85,B 0,C 180,E1 -22466.631,E2 -22466.631} C_VEL
LIN {X 0,Y 191.583,Z 533.979,A -85,B 0,C 180,E1 -22468.218,E2 -22468.218} C_VEL
LIN {X 0,Y 188.319,Z 530.123,A -85,B 0,C 180,E1 -22470.132,E2 -22470.132} C_VEL
LIN {X 0,Y 187.297,Z 528.48,A -85,B 0,C 180,E1 -22470.803,E2 -22470.803} C_VEL
LIN {X 0,Y 184.675,Z 525.987,A -85,B 0,C 180,E1 -22472.484,E2 -22472.484} C_VEL
LIN {X 0,Y 182.947,Z 523.09,A -85,B 0,C 180,E1 -22473.782,E2 -22473.782} C_VEL
LIN {X 0,Y 180.415,Z 521.37,A -85,B 0,C 180,E1 -22475.611,E2 -22475.611} C_VEL
LIN {X 0,Y 178.851,Z 518.842,A -85,B 0,C 180,E1 -22477.014,E2 -22477.014} C_VEL
LIN {X 0,Y 178.575,Z 517.669,A -85,B 0,C 180,E1 -22477.816,E2 -22477.816} C_VEL
LIN {X 0,Y 178.619,Z 517.329,A -85,B 0,C 180,E1 -22480.785,E2 -22480.785} C_VEL
LIN {X 0,Y 178.657,Z 517.313,A -85,B 0,C 180,E1 -22486.347,E2 -22486.347} C_VEL
LIN {X 0,Y 178.956,Z 517.309,A -85,B 0,C 180,E1 -22490.961,E2 -22490.961} C_VEL
LIN {X 0,Y 179.149,Z 517.288,A -85,B 0,C 180,E1 -22497.751,E2 -22497.751} C_VEL
LIN {X 0,Y 179.365,Z 517.233,A -85,B 0,C 180,E1 -22499.999,E2 -22499.999} C_VEL
LIN {X 0,Y 178.861,Z 517.301,A -85,B 0,C 180,E1 -22504.506,E2 -22504.506} C_VEL
LIN {X 0,Y 178.907,Z 517.281,A -85,B 0,C 180,E1 -22509.039,E2 -22509.039} C_VEL
LIN {X 0,Y 178.652,Z 517.357,A -85,B 0,C 180,E1 -22513.651,E2 -22513.651} C_VEL
LIN {X 0,Y 178.619,Z 517.331,A -85,B 0,C 180,E1 -22519.215,E2 -22519.215} C_VEL
LIN {X 0,Y 178.573,Z 517.627,A -85,B 0,C 180,E1 -22522.563,E2 -22522.563} C_VEL
LIN {X 0,Y 178.83,Z 518.758,A -85,B 0,C 180,E1 -22523.351,E2 -22523.351} C_VEL
LIN {X 0,Y 180.33,Z 521.243,A -85,B 0,C 180,E1 -22524.711,E2 -22524.711} C_VEL
LIN {X 0,Y 183.363,Z 523.652,A -85,B 0,C 180,E1 -22526.919,E2 -22526.919} C_VEL
LIN {X 0,Y 185.256,Z 526.752,A -85,B 0,C 180,E1 -22528.31,E2 -22528.31} C_VEL
LIN {X 0,Y 187.762,Z 529.072,A -85,B 0,C 180,E1 -22529.886,E2 -22529.886} C_VEL
LIN {X 0,Y 189.871,Z 532.223,A -85,B 0,C 180,E1 -22531.211,E2 -22531.211} C_VEL
LIN {X 0,Y 191.681,Z 534.105,A -85,B 0,C 180,E1 -22532.23,E2 -22532.23} C_VEL
LIN {X 0,Y 194.493,Z 537.902,A -85,B 0,C 180,E1 -22533.779,E2 -22533.779} C_VEL
LIN {X 0,Y 199.223,Z 544.352,A -85,B 0,C 180,E1 -22536.166,E2 -22536.166} C_VEL
LIN {X 0,Y 204.597,Z 552.191,A -85,B 0,C 180,E1 -22538.627,E2 -22538.627} C_VEL
LIN {X 0,Y 210.585,Z 561.692,A -85,B 0,C 180,E1 -22541.123,E2 -22541.123} C_VEL
LIN {X 0,Y 217.203,Z 573.412,A -85,B 0,C 180,E1 -22543.652,E2 -22543.652} C_VEL
LIN {X 0,Y 226.179,Z 590.562,A -85,B 0,C 180,E1 -22546.741,E2 -22546.741} C_VEL
LIN {X 0,Y 234.953,Z 603.794,A -85,B 0,C 180,E1 -22549.262,E2 -22549.262} C_VEL
LIN {X 0,Y 246.104,Z 617.434,A -85,B 0,C 180,E1 -22551.975,E2 -22551.975} C_VEL
LIN {X 0,Y 262.918,Z 634.4,A -85,B 0,C 180,E1 -22555.362,E2 -22555.362} C_VEL
LIN {X 0,Y 276.629,Z 646.347,A -85,B 0,C 180,E1 -22557.804,E2 -22557.804} C_VEL
LIN {X 0,Y 289.208,Z 656.261,A -85,B 0,C 180,E1 -22559.963,E2 -22559.963} C_VEL
LIN {X 0,Y 298.198,Z 663.283,A -85,B 0,C 180,E1 -22561.692,E2 -22561.692} C_VEL
LIN {X 0,Y 306.398,Z 669.463,A -85,B 0,C 180,E1 -22563.45,E2 -22563.45} C_VEL
LIN {X 0,Y 313.304,Z 674.516,A -85,B 0,C 180,E1 -22565.08,E2 -22565.08} C_VEL
LIN {X 0,Y 319.554,Z 679.105,A -85,B 0,C 180,E1 -22566.68,E2 -22566.68} C_VEL
LIN {X 0,Y 327.178,Z 684.48,A -85,B 0,C 180,E1 -22568.797,E2 -22568.797} C_VEL
LIN {X 0,Y 331.816,Z 687.577,A -85,B 0,C 180,E1 -22570.191,E2 -22570.191} C_VEL
LIN {X 0,Y 336.36,Z 690.986,A -85,B 0,C 180,E1 -22571.735,E2 -22571.735} C_VEL
LIN {X 0,Y 340.483,Z 693.757,A -85,B 0,C 180,E1 -22573.204,E2 -22573.204} C_VEL
LIN {X 0,Y 344.196,Z 695.859,A -85,B 0,C 180,E1 -22574.607,E2 -22574.607} C_VEL
LIN {X 0,Y 347.582,Z 698.012,A -85,B 0,C 180,E1 -22576.056,E2 -22576.056} C_VEL
LIN {X 0,Y 351.801,Z 701.179,A -85,B 0,C 180,E1 -22578.201,E2 -22578.201} C_VEL
LIN {X 0,Y 354.428,Z 702.897,A -85,B 0,C 180,E1 -22579.72,E2 -22579.72} C_VEL
LIN {X 0,Y 356.329,Z 703.927,A -85,B 0,C 180,E1 -22580.922,E2 -22580.922} C_VEL
LIN {X 0,Y 359.403,Z 705.503,A -85,B 0,C 180,E1 -22583.262,E2 -22583.262} C_VEL
LIN {X 0,Y 361.593,Z 706.408,A -85,B 0,C 180,E1 -22585.541,E2 -22585.541} C_VEL
